ABB RAPID module: P6.mod

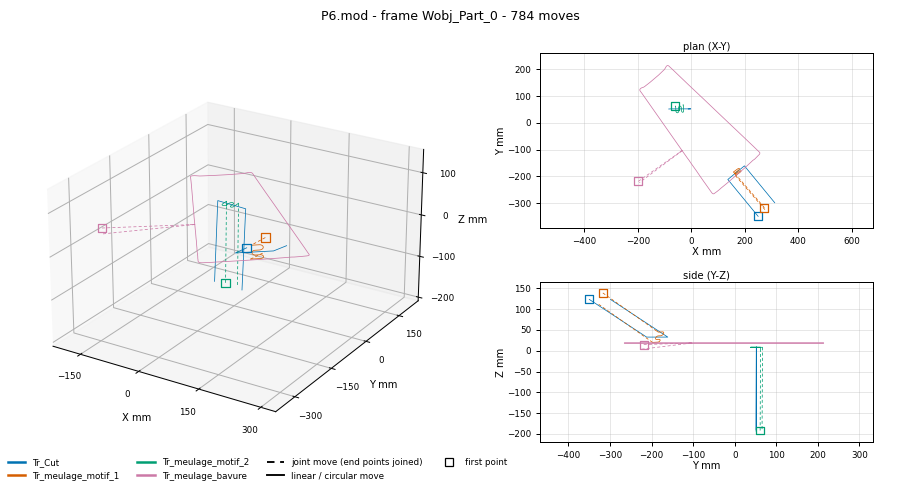
[picture p0: tool path of P6.mod in frame Wobj_Part_0, 784 of 794 moves have a stored position in this frame; points joined in program order, loops and branches not executed]
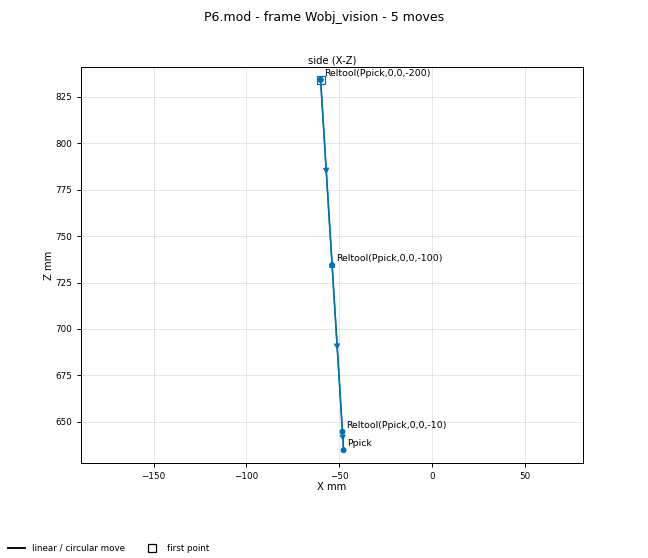
[picture p1: tool path of P6.mod in frame Wobj_vision, 5 of 794 moves have a stored position in this frame; points joined in program order, loops and branches not executed]
MODULE P6
	LOCAL CONST Speeddata vitesse_Tronconnage :=[10, 500, 0, 0];
	LOCAL CONST Robtarget Coupe_0 :=[[171.071296875,-183.16509375,32.79853125],[0.442625876519456,0.144946358690586,0.692091434062249,0.551436608718884],[0,0,0,0],[8.999999E+09,8.999999E+09,8.999999E+09,8.999999E+09,8.999999E+09,8.999999E+09]];
	LOCAL CONST Robtarget Coupe_1 :=[[-43.76221875,52.00546875,8.2563916015625],[0.723189251048334,-0.000890046614138083,-0.690648714177327,0.00093198196284652],[0,0,0,0],[8.999999E+09,8.999999E+09,8.999999E+09,8.999999E+09,8.999999E+09,8.999999E+09]];
	LOCAL CONST Robtarget Tr_meulage_motif_1_App1 :=[[272.919270252157,-317.055343641232,138.932114514029],[0.481869465480674,-0.803479210242735,-0.299818873825779,0.179809954793727],[0,0,0,0],[8.999999E+09,8.999999E+09,8.999999E+09,8.999999E+09,8.999999E+09,8.999999E+09]];
	LOCAL CONST Robtarget Tr_meulage_motif_1_App2 :=[[163.119364293858,-190.415905463312,49.4534391241389],[0.481869465480674,-0.803479210242735,-0.299818873825779,0.179809954793727],[0,0,0,0],[8.999999E+09,8.999999E+09,8.999999E+09,8.999999E+09,8.999999E+09,8.999999E+09]];
	LOCAL CONST Robtarget Tr_meulage_motif_1_P0 :=[[157.340421875,-183.750671875,44.74403515625],[0.481869465480674,-0.803479210242735,-0.299818873825779,0.179809954793727],[0,0,0,0],[8.999999E+09,8.999999E+09,8.999999E+09,8.999999E+09,8.999999E+09,8.999999E+09]];
	LOCAL CONST Robtarget Tr_meulage_motif_1_P1 :=[[158.144921875,-183.157578125,44.775765625],[0.481869465480674,-0.803479210242735,-0.299818873825779,0.179809954793727],[0,0,0,0],[8.999999E+09,8.999999E+09,8.999999E+09,8.999999E+09,8.999999E+09,8.999999E+09]];
	LOCAL CONST Robtarget Tr_meulage_motif_1_P2 :=[[158.949421875,-182.56446875,44.80749609375],[0.481869465480674,-0.803479210242735,-0.299818873825779,0.179809954793727],[0,0,0,0],[8.999999E+09,8.999999E+09,8.999999E+09,8.999999E+09,8.999999E+09,8.999999E+09]];
	LOCAL CONST Robtarget Tr_meulage_motif_1_P3 :=[[159.753921875,-181.971359375,44.8392265625],[0.481869465480674,-0.803479210242735,-0.299818873825779,0.179809954793727],[0,0,0,0],[8.999999E+09,8.999999E+09,8.999999E+09,8.999999E+09,8.999999E+09,8.999999E+09]];
	LOCAL CONST Robtarget Tr_meulage_motif_1_P4 :=[[160.558421875,-181.37825,44.87095703125],[0.481869465480674,-0.803479210242735,-0.299818873825779,0.179809954793727],[0,0,0,0],[8.999999E+09,8.999999E+09,8.999999E+09,8.999999E+09,8.999999E+09,8.999999E+09]];
	LOCAL CONST Robtarget Tr_meulage_motif_1_P5 :=[[161.362921875,-180.78515625,44.9026875],[0.481869465480674,-0.803479210242735,-0.299818873825779,0.179809954793727],[0,0,0,0],[8.999999E+09,8.999999E+09,8.999999E+09,8.999999E+09,8.999999E+09,8.999999E+09]];
	LOCAL CONST Robtarget Tr_meulage_motif_1_P6 :=[[162.167421875,-180.192046875,44.93441796875],[0.481869465480674,-0.803479210242735,-0.299818873825779,0.179809954793727],[0,0,0,0],[8.999999E+09,8.999999E+09,8.999999E+09,8.999999E+09,8.999999E+09,8.999999E+09]];
	LOCAL CONST Robtarget Tr_meulage_motif_1_P7 :=[[162.971921875,-179.5989375,44.9661484375],[0.481869465480674,-0.803479210242735,-0.299818873825779,0.179809954793727],[0,0,0,0],[8.999999E+09,8.999999E+09,8.999999E+09,8.999999E+09,8.999999E+09,8.999999E+09]];
	LOCAL CONST Robtarget Tr_meulage_motif_1_P8 :=[[163.776421875,-179.005828125,44.99787890625],[0.481869465480674,-0.803479210242735,-0.299818873825779,0.179809954793727],[0,0,0,0],[8.999999E+09,8.999999E+09,8.999999E+09,8.999999E+09,8.999999E+09,8.999999E+09]];
	LOCAL CONST Robtarget Tr_meulage_motif_1_P9 :=[[164.580921875,-178.412734375,45.029609375],[0.481869465480674,-0.803479210242735,-0.299818873825779,0.179809954793727],[0,0,0,0],[8.999999E+09,8.999999E+09,8.999999E+09,8.999999E+09,8.999999E+09,8.999999E+09]];
	LOCAL CONST Robtarget Tr_meulage_motif_1_P10 :=[[165.385421875,-177.819625,45.06133984375],[0.481869465480674,-0.803479210242735,-0.299818873825779,0.179809954793727],[0,0,0,0],[8.999999E+09,8.999999E+09,8.999999E+09,8.999999E+09,8.999999E+09,8.999999E+09]];
	LOCAL CONST Robtarget Tr_meulage_motif_1_P11 :=[[166.189921875,-177.226515625,45.0930703125],[0.481869465480674,-0.803479210242735,-0.299818873825779,0.179809954793727],[0,0,0,0],[8.999999E+09,8.999999E+09,8.999999E+09,8.999999E+09,8.999999E+09,8.999999E+09]];
	LOCAL CONST Robtarget Tr_meulage_motif_1_P12 :=[[166.994421875,-176.633421875,45.12480078125],[0.481869465480674,-0.803479210242735,-0.299818873825779,0.179809954793727],[0,0,0,0],[8.999999E+09,8.999999E+09,8.999999E+09,8.999999E+09,8.999999E+09,8.999999E+09]];
	LOCAL CONST Robtarget Tr_meulage_motif_1_P13 :=[[167.798921875,-176.0403125,45.15653125],[0.481869465480674,-0.803479210242735,-0.299818873825779,0.179809954793727],[0,0,0,0],[8.999999E+09,8.999999E+09,8.999999E+09,8.999999E+09,8.999999E+09,8.999999E+09]];
	LOCAL CONST Robtarget Tr_meulage_motif_1_P14 :=[[168.603421875,-175.447203125,45.18826171875],[0.481869465480674,-0.803479210242735,-0.299818873825779,0.179809954793727],[0,0,0,0],[8.999999E+09,8.999999E+09,8.999999E+09,8.999999E+09,8.999999E+09,8.999999E+09]];
	LOCAL CONST Robtarget Tr_meulage_motif_1_P15 :=[[169.407921875,-174.85409375,45.2199921875],[0.481869465480674,-0.803479210242735,-0.299818873825779,0.179809954793727],[0,0,0,0],[8.999999E+09,8.999999E+09,8.999999E+09,8.999999E+09,8.999999E+09,8.999999E+09]];
	LOCAL CONST Robtarget Tr_meulage_motif_1_P16 :=[[170.212421875,-174.261,45.25172265625],[0.481869465480674,-0.803479210242735,-0.299818873825779,0.179809954793727],[0,0,0,0],[8.999999E+09,8.999999E+09,8.999999E+09,8.999999E+09,8.999999E+09,8.999999E+09]];
	LOCAL CONST Robtarget Tr_meulage_motif_1_P17 :=[[171.016921875,-173.667890625,45.28345703125],[0.481869465480674,-0.803479210242735,-0.299818873825779,0.179809954793727],[0,0,0,0],[8.999999E+09,8.999999E+09,8.999999E+09,8.999999E+09,8.999999E+09,8.999999E+09]];
	LOCAL CONST Robtarget Tr_meulage_motif_1_P18 :=[[171.821421875,-173.07478125,45.3151875],[0.481869465480674,-0.803479210242735,-0.299818873825779,0.179809954793727],[0,0,0,0],[8.999999E+09,8.999999E+09,8.999999E+09,8.999999E+09,8.999999E+09,8.999999E+09]];
	LOCAL CONST Robtarget Tr_meulage_motif_1_P19 :=[[172.657078125,-172.531453125,45.25290625],[0.481869465480674,-0.803479210242735,-0.299818873825779,0.179809954793727],[0,0,0,0],[8.999999E+09,8.999999E+09,8.999999E+09,8.999999E+09,8.999999E+09,8.999999E+09]];
	LOCAL CONST Robtarget Tr_meulage_motif_1_P20 :=[[173.489453125,-172.0566875,45.1038671875],[0.481869465480674,-0.803479210242735,-0.299818873825779,0.179809954793727],[0,0,0,0],[8.999999E+09,8.999999E+09,8.999999E+09,8.999999E+09,8.999999E+09,8.999999E+09]];
	LOCAL CONST Robtarget Tr_meulage_motif_1_P21 :=[[174.26675,-171.6624375,44.90041796875],[0.481869465480674,-0.803479210242735,-0.299818873825779,0.179809954793727],[0,0,0,0],[8.999999E+09,8.999999E+09,8.999999E+09,8.999999E+09,8.999999E+09,8.999999E+09]];
	LOCAL CONST Robtarget Tr_meulage_motif_1_P22 :=[[174.96275,-171.330828125,44.69023828125],[0.481869465480674,-0.803479210242735,-0.299818873825779,0.179809954793727],[0,0,0,0],[8.999999E+09,8.999999E+09,8.999999E+09,8.999999E+09,8.999999E+09,8.999999E+09]];
	LOCAL CONST Robtarget Tr_meulage_motif_1_P23 :=[[176.05546875,-170.9305,44.2027421875],[0.481869465480674,-0.803479210242735,-0.299818873825779,0.179809954793727],[0,0,0,0],[8.999999E+09,8.999999E+09,8.999999E+09,8.999999E+09,8.999999E+09,8.999999E+09]];
	LOCAL CONST Robtarget Tr_meulage_motif_1_P24 :=[[177.16384375,-170.67090625,43.5164765625],[0.481869465480674,-0.803479210242735,-0.299818873825779,0.179809954793727],[0,0,0,0],[8.999999E+09,8.999999E+09,8.999999E+09,8.999999E+09,8.999999E+09,8.999999E+09]];
	LOCAL CONST Robtarget Tr_meulage_motif_1_P25 :=[[178.189625,-170.588109375,42.67519921875],[0.481869465480674,-0.803479210242735,-0.299818873825779,0.179809954793727],[0,0,0,0],[8.999999E+09,8.999999E+09,8.999999E+09,8.999999E+09,8.999999E+09,8.999999E+09]];
	LOCAL CONST Robtarget Tr_meulage_motif_1_P26 :=[[178.9571875,-170.756390625,41.74423828125],[0.481869465480674,-0.803479210242735,-0.299818873825779,0.179809954793727],[0,0,0,0],[8.999999E+09,8.999999E+09,8.999999E+09,8.999999E+09,8.999999E+09,8.999999E+09]];
	LOCAL CONST Robtarget Tr_meulage_motif_1_P27 :=[[179.2126875,-171.025796875,41.1549609375],[0.481869465480674,-0.803479210242735,-0.299818873825779,0.179809954793727],[0,0,0,0],[8.999999E+09,8.999999E+09,8.999999E+09,8.999999E+09,8.999999E+09,8.999999E+09]];
	LOCAL CONST Robtarget Tr_meulage_motif_1_P28 :=[[179.43475,-171.297015625,40.594265625],[0.481869465480674,-0.803479210242735,-0.299818873825779,0.179809954793727],[0,0,0,0],[8.999999E+09,8.999999E+09,8.999999E+09,8.999999E+09,8.999999E+09,8.999999E+09]];
	LOCAL CONST Robtarget Tr_meulage_motif_1_P29 :=[[179.612625,-171.60071875,40.03196484375],[0.481869465480674,-0.803479210242735,-0.299818873825779,0.179809954793727],[0,0,0,0],[8.999999E+09,8.999999E+09,8.999999E+09,8.999999E+09,8.999999E+09,8.999999E+09]];
	LOCAL CONST Robtarget Tr_meulage_motif_1_P30 :=[[179.5818125,-172.348109375,39.0819453125],[0.481869465480674,-0.803479210242735,-0.299818873825779,0.179809954793727],[0,0,0,0],[8.999999E+09,8.999999E+09,8.999999E+09,8.999999E+09,8.999999E+09,8.999999E+09]];
	LOCAL CONST Robtarget Tr_meulage_motif_1_P31 :=[[179.230703125,-173.2690625,38.20121484375],[0.481869465480674,-0.803479210242735,-0.299818873825779,0.179809954793727],[0,0,0,0],[8.999999E+09,8.999999E+09,8.999999E+09,8.999999E+09,8.999999E+09,8.999999E+09]];
	LOCAL CONST Robtarget Tr_meulage_motif_1_P32 :=[[178.685734375,-174.216015625,37.4659140625],[0.481869465480674,-0.803479210242735,-0.299818873825779,0.179809954793727],[0,0,0,0],[8.999999E+09,8.999999E+09,8.999999E+09,8.999999E+09,8.999999E+09,8.999999E+09]];
	LOCAL CONST Robtarget Tr_meulage_motif_1_P33 :=[[178.265875,-174.785859375,37.10854296875],[0.481869465480674,-0.803479210242735,-0.299818873825779,0.179809954793727],[0,0,0,0],[8.999999E+09,8.999999E+09,8.999999E+09,8.999999E+09,8.999999E+09,8.999999E+09]];
	LOCAL CONST Robtarget Tr_meulage_motif_1_P34 :=[[177.497859375,-175.672734375,36.6583984375],[0.481869465480674,-0.803479210242735,-0.299818873825779,0.179809954793727],[0,0,0,0],[8.999999E+09,8.999999E+09,8.999999E+09,8.999999E+09,8.999999E+09,8.999999E+09]];
	LOCAL CONST Robtarget Tr_meulage_motif_1_P35 :=[[176.906734375,-176.28225,36.40765234375],[0.481869465480674,-0.803479210242735,-0.299818873825779,0.179809954793727],[0,0,0,0],[8.999999E+09,8.999999E+09,8.999999E+09,8.999999E+09,8.999999E+09,8.999999E+09]];
	LOCAL CONST Robtarget Tr_meulage_motif_1_P36 :=[[176.22559375,-176.918890625,36.204703125],[0.481869465480674,-0.803479210242735,-0.299818873825779,0.179809954793727],[0,0,0,0],[8.999999E+09,8.999999E+09,8.999999E+09,8.999999E+09,8.999999E+09,8.999999E+09]];
	LOCAL CONST Robtarget Tr_meulage_motif_1_P37 :=[[175.47240625,-177.54559375,36.08148046875],[0.481869465480674,-0.803479210242735,-0.299818873825779,0.179809954793727],[0,0,0,0],[8.999999E+09,8.999999E+09,8.999999E+09,8.999999E+09,8.999999E+09,8.999999E+09]];
	LOCAL CONST Robtarget Tr_meulage_motif_1_P38 :=[[174.71103125,-178.17965625,35.95620703125],[0.481869465480674,-0.803479210242735,-0.299818873825779,0.179809954793727],[0,0,0,0],[8.999999E+09,8.999999E+09,8.999999E+09,8.999999E+09,8.999999E+09,8.999999E+09]];
	LOCAL CONST Robtarget Tr_meulage_motif_1_P39 :=[[173.90653125,-178.77275,35.9244765625],[0.481869465480674,-0.803479210242735,-0.299818873825779,0.179809954793727],[0,0,0,0],[8.999999E+09,8.999999E+09,8.999999E+09,8.999999E+09,8.999999E+09,8.999999E+09]];
	LOCAL CONST Robtarget Tr_meulage_motif_1_P40 :=[[173.10203125,-179.365859375,35.89274609375],[0.481869465480674,-0.803479210242735,-0.299818873825779,0.179809954793727],[0,0,0,0],[8.999999E+09,8.999999E+09,8.999999E+09,8.999999E+09,8.999999E+09,8.999999E+09]];
	LOCAL CONST Robtarget Tr_meulage_motif_1_P41 :=[[172.29753125,-179.95896875,35.861015625],[0.481869465480674,-0.803479210242735,-0.299818873825779,0.179809954793727],[0,0,0,0],[8.999999E+09,8.999999E+09,8.999999E+09,8.999999E+09,8.999999E+09,8.999999E+09]];
	LOCAL CONST Robtarget Tr_meulage_motif_1_P42 :=[[171.49303125,-180.552078125,35.82928515625],[0.481869465480674,-0.803479210242735,-0.299818873825779,0.179809954793727],[0,0,0,0],[8.999999E+09,8.999999E+09,8.999999E+09,8.999999E+09,8.999999E+09,8.999999E+09]];
	LOCAL CONST Robtarget Tr_meulage_motif_1_P43 :=[[170.68853125,-181.145171875,35.7975546875],[0.481869465480674,-0.803479210242735,-0.299818873825779,0.179809954793727],[0,0,0,0],[8.999999E+09,8.999999E+09,8.999999E+09,8.999999E+09,8.999999E+09,8.999999E+09]];
	LOCAL CONST Robtarget Tr_meulage_motif_1_P44 :=[[169.88403125,-181.73828125,35.76582421875],[0.481869465480674,-0.803479210242735,-0.299818873825779,0.179809954793727],[0,0,0,0],[8.999999E+09,8.999999E+09,8.999999E+09,8.999999E+09,8.999999E+09,8.999999E+09]];
	LOCAL CONST Robtarget Tr_meulage_motif_1_P45 :=[[169.07953125,-182.331390625,35.73409375],[0.481869465480674,-0.803479210242735,-0.299818873825779,0.179809954793727],[0,0,0,0],[8.999999E+09,8.999999E+09,8.999999E+09,8.999999E+09,8.999999E+09,8.999999E+09]];
	LOCAL CONST Robtarget Tr_meulage_motif_1_P46 :=[[168.27503125,-182.9245,35.70236328125],[0.481869465480674,-0.803479210242735,-0.299818873825779,0.179809954793727],[0,0,0,0],[8.999999E+09,8.999999E+09,8.999999E+09,8.999999E+09,8.999999E+09,8.999999E+09]];
	LOCAL CONST Robtarget Tr_meulage_motif_1_P47 :=[[167.47053125,-183.51759375,35.6706328125],[0.481869465480674,-0.803479210242735,-0.299818873825779,0.179809954793727],[0,0,0,0],[8.999999E+09,8.999999E+09,8.999999E+09,8.999999E+09,8.999999E+09,8.999999E+09]];
	LOCAL CONST Robtarget Tr_meulage_motif_1_P48 :=[[166.66603125,-184.110703125,35.63890234375],[0.481869465480674,-0.803479210242735,-0.299818873825779,0.179809954793727],[0,0,0,0],[8.999999E+09,8.999999E+09,8.999999E+09,8.999999E+09,8.999999E+09,8.999999E+09]];
	LOCAL CONST Robtarget Tr_meulage_motif_1_P49 :=[[165.90465625,-184.744765625,35.51362890625],[0.481869465480674,-0.803479210242735,-0.299818873825779,0.179809954793727],[0,0,0,0],[8.999999E+09,8.999999E+09,8.999999E+09,8.999999E+09,8.999999E+09,8.999999E+09]];
	LOCAL CONST Robtarget Tr_meulage_motif_1_P50 :=[[165.214125,-185.39275,35.3045234375],[0.481869465480674,-0.803479210242735,-0.299818873825779,0.179809954793727],[0,0,0,0],[8.999999E+09,8.999999E+09,8.999999E+09,8.999999E+09,8.999999E+09,8.999999E+09]];
	LOCAL CONST Robtarget Tr_meulage_motif_1_P51 :=[[164.61940625,-186.01,35.0469609375],[0.481869465480674,-0.803479210242735,-0.299818873825779,0.179809954793727],[0,0,0,0],[8.999999E+09,8.999999E+09,8.999999E+09,8.999999E+09,8.999999E+09,8.999999E+09]];
	LOCAL CONST Robtarget Tr_meulage_motif_1_P52 :=[[164.149140625,-186.55675,34.76648046875],[0.481869465480674,-0.803479210242735,-0.299818873825779,0.179809954793727],[0,0,0,0],[8.999999E+09,8.999999E+09,8.999999E+09,8.999999E+09,8.999999E+09,8.999999E+09]];
	LOCAL CONST Robtarget Tr_meulage_motif_1_P53 :=[[163.539421875,-187.442046875,34.171875],[0.481869465480674,-0.803479210242735,-0.299818873825779,0.179809954793727],[0,0,0,0],[8.999999E+09,8.999999E+09,8.999999E+09,8.999999E+09,8.999999E+09,8.999999E+09]];
	LOCAL CONST Robtarget Tr_meulage_motif_1_P54 :=[[163.116703125,-188.346921875,33.3784765625],[0.481869465480674,-0.803479210242735,-0.299818873825779,0.179809954793727],[0,0,0,0],[8.999999E+09,8.999999E+09,8.999999E+09,8.999999E+09,8.999999E+09,8.999999E+09]];
	LOCAL CONST Robtarget Tr_meulage_motif_1_P55 :=[[163.037609375,-189.093265625,32.4745390625],[0.481869465480674,-0.803479210242735,-0.299818873825779,0.179809954793727],[0,0,0,0],[8.999999E+09,8.999999E+09,8.999999E+09,8.999999E+09,8.999999E+09,8.999999E+09]];
	LOCAL CONST Robtarget Tr_meulage_motif_1_P56 :=[[163.12175,-189.4871875,31.880873046875],[0.481869465480674,-0.803479210242735,-0.299818873825779,0.179809954793727],[0,0,0,0],[8.999999E+09,8.999999E+09,8.999999E+09,8.999999E+09,8.999999E+09,8.999999E+09]];
	LOCAL CONST Robtarget Tr_meulage_motif_1_P57 :=[[163.328984375,-189.840875,31.225939453125],[0.481869465480674,-0.803479210242735,-0.299818873825779,0.179809954793727],[0,0,0,0],[8.999999E+09,8.999999E+09,8.999999E+09,8.999999E+09,8.999999E+09,8.999999E+09]];
	LOCAL CONST Robtarget Tr_meulage_motif_1_P58 :=[[163.641375,-190.116953125,30.57526171875],[0.481869465480674,-0.803479210242735,-0.299818873825779,0.179809954793727],[0,0,0,0],[8.999999E+09,8.999999E+09,8.999999E+09,8.999999E+09,8.999999E+09,8.999999E+09]];
	LOCAL CONST Robtarget Tr_meulage_motif_1_P59 :=[[164.351125,-190.322640625,29.648857421875],[0.481869465480674,-0.803479210242735,-0.299818873825779,0.179809954793727],[0,0,0,0],[8.999999E+09,8.999999E+09,8.999999E+09,8.999999E+09,8.999999E+09,8.999999E+09]];
	LOCAL CONST Robtarget Tr_meulage_motif_1_P60 :=[[164.881125,-190.317140625,29.165380859375],[0.481869465480674,-0.803479210242735,-0.299818873825779,0.179809954793727],[0,0,0,0],[8.999999E+09,8.999999E+09,8.999999E+09,8.999999E+09,8.999999E+09,8.999999E+09]];
	LOCAL CONST Robtarget Tr_meulage_motif_1_P61 :=[[165.892734375,-190.15484375,28.44130859375],[0.481869465480674,-0.803479210242735,-0.299818873825779,0.179809954793727],[0,0,0,0],[8.999999E+09,8.999999E+09,8.999999E+09,8.999999E+09,8.999999E+09,8.999999E+09]];
	LOCAL CONST Robtarget Tr_meulage_motif_1_P62 :=[[166.5030625,-189.97740625,28.108583984375],[0.481869465480674,-0.803479210242735,-0.299818873825779,0.179809954793727],[0,0,0,0],[8.999999E+09,8.999999E+09,8.999999E+09,8.999999E+09,8.999999E+09,8.999999E+09]];
	LOCAL CONST Robtarget Tr_meulage_motif_1_P63 :=[[167.585140625,-189.53753125,27.682701171875],[0.481869465480674,-0.803479210242735,-0.299818873825779,0.179809954793727],[0,0,0,0],[8.999999E+09,8.999999E+09,8.999999E+09,8.999999E+09,8.999999E+09,8.999999E+09]];
	LOCAL CONST Robtarget Tr_meulage_motif_1_P64 :=[[168.3485625,-189.169078125,27.458333984375],[0.481869465480674,-0.803479210242735,-0.299818873825779,0.179809954793727],[0,0,0,0],[8.999999E+09,8.999999E+09,8.999999E+09,8.999999E+09,8.999999E+09,8.999999E+09]];
	LOCAL CONST Robtarget Tr_meulage_motif_1_P65 :=[[169.16703125,-188.70015625,27.31453125],[0.481869465480674,-0.803479210242735,-0.299818873825779,0.179809954793727],[0,0,0,0],[8.999999E+09,8.999999E+09,8.999999E+09,8.999999E+09,8.999999E+09,8.999999E+09]];
	LOCAL CONST Robtarget Tr_meulage_motif_1_P66 :=[[169.99315625,-188.16253125,27.25359765625],[0.481869465480674,-0.803479210242735,-0.299818873825779,0.179809954793727],[0,0,0,0],[8.999999E+09,8.999999E+09,8.999999E+09,8.999999E+09,8.999999E+09,8.999999E+09]];
	LOCAL CONST Robtarget Tr_meulage_motif_1_P67 :=[[170.8288125,-187.619203125,27.19131640625],[0.481869465480674,-0.803479210242735,-0.299818873825779,0.179809954793727],[0,0,0,0],[8.999999E+09,8.999999E+09,8.999999E+09,8.999999E+09,8.999999E+09,8.999999E+09]];
	LOCAL CONST Robtarget Tr_meulage_motif_1_P68 :=[[171.6333125,-187.02609375,27.223046875],[0.481869465480674,-0.803479210242735,-0.299818873825779,0.179809954793727],[0,0,0,0],[8.999999E+09,8.999999E+09,8.999999E+09,8.999999E+09,8.999999E+09,8.999999E+09]];
	LOCAL CONST Robtarget Tr_meulage_motif_1_P69 :=[[172.4378125,-186.432984375,27.25477734375],[0.481869465480674,-0.803479210242735,-0.299818873825779,0.179809954793727],[0,0,0,0],[8.999999E+09,8.999999E+09,8.999999E+09,8.999999E+09,8.999999E+09,8.999999E+09]];
	LOCAL CONST Robtarget Tr_meulage_motif_1_P70 :=[[173.2423125,-185.839890625,27.2865078125],[0.481869465480674,-0.803479210242735,-0.299818873825779,0.179809954793727],[0,0,0,0],[8.999999E+09,8.999999E+09,8.999999E+09,8.999999E+09,8.999999E+09,8.999999E+09]];
	LOCAL CONST Robtarget Tr_meulage_motif_1_P71 :=[[174.0468125,-185.24678125,27.31823828125],[0.481869465480674,-0.803479210242735,-0.299818873825779,0.179809954793727],[0,0,0,0],[8.999999E+09,8.999999E+09,8.999999E+09,8.999999E+09,8.999999E+09,8.999999E+09]];
	LOCAL CONST Robtarget Tr_meulage_motif_1_P72 :=[[174.8513125,-184.653671875,27.34996875],[0.481869465480674,-0.803479210242735,-0.299818873825779,0.179809954793727],[0,0,0,0],[8.999999E+09,8.999999E+09,8.999999E+09,8.999999E+09,8.999999E+09,8.999999E+09]];
	LOCAL CONST Robtarget Tr_meulage_motif_1_P73 :=[[175.6558125,-184.0605625,27.38169921875],[0.481869465480674,-0.803479210242735,-0.299818873825779,0.179809954793727],[0,0,0,0],[8.999999E+09,8.999999E+09,8.999999E+09,8.999999E+09,8.999999E+09,8.999999E+09]];
	LOCAL CONST Robtarget Tr_meulage_motif_1_P74 :=[[176.4603125,-183.46746875,27.413431640625],[0.481869465480674,-0.803479210242735,-0.299818873825779,0.179809954793727],[0,0,0,0],[8.999999E+09,8.999999E+09,8.999999E+09,8.999999E+09,8.999999E+09,8.999999E+09]];
	LOCAL CONST Robtarget Tr_meulage_motif_1_P75 :=[[177.2648125,-182.874359375,27.445162109375],[0.481869465480674,-0.803479210242735,-0.299818873825779,0.179809954793727],[0,0,0,0],[8.999999E+09,8.999999E+09,8.999999E+09,8.999999E+09,8.999999E+09,8.999999E+09]];
	LOCAL CONST Robtarget Tr_meulage_motif_1_P76 :=[[178.0693125,-182.28125,27.476892578125],[0.481869465480674,-0.803479210242735,-0.299818873825779,0.179809954793727],[0,0,0,0],[8.999999E+09,8.999999E+09,8.999999E+09,8.999999E+09,8.999999E+09,8.999999E+09]];
	LOCAL CONST Robtarget Tr_meulage_motif_1_P77 :=[[178.8738125,-181.688140625,27.508623046875],[0.481869465480674,-0.803479210242735,-0.299818873825779,0.179809954793727],[0,0,0,0],[8.999999E+09,8.999999E+09,8.999999E+09,8.999999E+09,8.999999E+09,8.999999E+09]];
	LOCAL CONST Robtarget Tr_meulage_motif_1_P78 :=[[179.70946875,-181.1448125,27.446341796875],[0.481869465480674,-0.803479210242735,-0.299818873825779,0.179809954793727],[0,0,0,0],[8.999999E+09,8.999999E+09,8.999999E+09,8.999999E+09,8.999999E+09,8.999999E+09]];
	LOCAL CONST Robtarget Tr_meulage_motif_1_P79 :=[[180.54184375,-180.6700625,27.297302734375],[0.481869465480674,-0.803479210242735,-0.299818873825779,0.179809954793727],[0,0,0,0],[8.999999E+09,8.999999E+09,8.999999E+09,8.999999E+09,8.999999E+09,8.999999E+09]];
	LOCAL CONST Robtarget Tr_meulage_motif_1_P80 :=[[181.31915625,-180.2758125,27.09385546875],[0.481869465480674,-0.803479210242735,-0.299818873825779,0.179809954793727],[0,0,0,0],[8.999999E+09,8.999999E+09,8.999999E+09,8.999999E+09,8.999999E+09,8.999999E+09]];
	LOCAL CONST Robtarget Tr_meulage_motif_1_P81 :=[[182.015140625,-179.9441875,26.883673828125],[0.481869465480674,-0.803479210242735,-0.299818873825779,0.179809954793727],[0,0,0,0],[8.999999E+09,8.999999E+09,8.999999E+09,8.999999E+09,8.999999E+09,8.999999E+09]];
	LOCAL CONST Robtarget Tr_meulage_motif_1_P82 :=[[183.107859375,-179.543859375,26.3961796875],[0.481869465480674,-0.803479210242735,-0.299818873825779,0.179809954793727],[0,0,0,0],[8.999999E+09,8.999999E+09,8.999999E+09,8.999999E+09,8.999999E+09,8.999999E+09]];
	LOCAL CONST Robtarget Tr_meulage_motif_1_P83 :=[[184.177765625,-179.34309375,25.668513671875],[0.481869465480674,-0.803479210242735,-0.299818873825779,0.179809954793727],[0,0,0,0],[8.999999E+09,8.999999E+09,8.999999E+09,8.999999E+09,8.999999E+09,8.999999E+09]];
	LOCAL CONST Robtarget Tr_meulage_motif_1_P84 :=[[185.032515625,-179.42725,24.76698828125],[0.481869465480674,-0.803479210242735,-0.299818873825779,0.179809954793727],[0,0,0,0],[8.999999E+09,8.999999E+09,8.999999E+09,8.999999E+09,8.999999E+09,8.999999E+09]];
	LOCAL CONST Robtarget Tr_meulage_motif_1_P85 :=[[185.499296875,-179.730578125,23.937677734375],[0.481869465480674,-0.803479210242735,-0.299818873825779,0.179809954793727],[0,0,0,0],[8.999999E+09,8.999999E+09,8.999999E+09,8.999999E+09,8.999999E+09,8.999999E+09]];
	LOCAL CONST Robtarget Tr_meulage_motif_1_P86 :=[[185.462265625,-179.8925,23.759970703125],[0.481869465480674,-0.803479210242735,-0.299818873825779,0.179809954793727],[0,0,0,0],[8.999999E+09,8.999999E+09,8.999999E+09,8.999999E+09,8.999999E+09,8.999999E+09]];
	LOCAL CONST Robtarget Tr_meulage_motif_1_P87 :=[[185.606953125,-180.263609375,23.14011328125],[0.481869465480674,-0.803479210242735,-0.299818873825779,0.179809954793727],[0,0,0,0],[8.999999E+09,8.999999E+09,8.999999E+09,8.999999E+09,8.999999E+09,8.999999E+09]];
	LOCAL CONST Robtarget Tr_meulage_motif_1_P88 :=[[185.371328125,-181.053578125,22.3239765625],[0.481869465480674,-0.803479210242735,-0.299818873825779,0.179809954793727],[0,0,0,0],[8.999999E+09,8.999999E+09,8.999999E+09,8.999999E+09,8.999999E+09,8.999999E+09]];
	LOCAL CONST Robtarget Tr_meulage_motif_1_P89 :=[[185.07846875,-181.574546875,21.913001953125],[0.481869465480674,-0.803479210242735,-0.299818873825779,0.179809954793727],[0,0,0,0],[8.999999E+09,8.999999E+09,8.999999E+09,8.999999E+09,8.999999E+09,8.999999E+09]];
	LOCAL CONST Robtarget Tr_meulage_motif_1_P90 :=[[184.34728125,-182.462515625,21.427361328125],[0.481869465480674,-0.803479210242735,-0.299818873825779,0.179809954793727],[0,0,0,0],[8.999999E+09,8.999999E+09,8.999999E+09,8.999999E+09,8.999999E+09,8.999999E+09]];
	LOCAL CONST Robtarget Tr_meulage_motif_1_P91 :=[[183.756140625,-183.072015625,21.176615234375],[0.481869465480674,-0.803479210242735,-0.299818873825779,0.179809954793727],[0,0,0,0],[8.999999E+09,8.999999E+09,8.999999E+09,8.999999E+09,8.999999E+09,8.999999E+09]];
	LOCAL CONST Robtarget Tr_meulage_motif_1_P92 :=[[183.075015625,-183.70865625,20.973666015625],[0.481869465480674,-0.803479210242735,-0.299818873825779,0.179809954793727],[0,0,0,0],[8.999999E+09,8.999999E+09,8.999999E+09,8.999999E+09,8.999999E+09,8.999999E+09]];
	LOCAL CONST Robtarget Tr_meulage_motif_1_P93 :=[[182.3218125,-184.335375,20.85044140625],[0.481869465480674,-0.803479210242735,-0.299818873825779,0.179809954793727],[0,0,0,0],[8.999999E+09,8.999999E+09,8.999999E+09,8.999999E+09,8.999999E+09,8.999999E+09]];
	LOCAL CONST Robtarget Tr_meulage_motif_1_P94 :=[[181.5604375,-184.969421875,20.725169921875],[0.481869465480674,-0.803479210242735,-0.299818873825779,0.179809954793727],[0,0,0,0],[8.999999E+09,8.999999E+09,8.999999E+09,8.999999E+09,8.999999E+09,8.999999E+09]];
	LOCAL CONST Robtarget Tr_meulage_motif_1_P95 :=[[180.7559375,-185.56253125,20.693439453125],[0.481869465480674,-0.803479210242735,-0.299818873825779,0.179809954793727],[0,0,0,0],[8.999999E+09,8.999999E+09,8.999999E+09,8.999999E+09,8.999999E+09,8.999999E+09]];
	LOCAL CONST Robtarget Tr_meulage_motif_1_P96 :=[[179.9514375,-186.155640625,20.661708984375],[0.481869465480674,-0.803479210242735,-0.299818873825779,0.179809954793727],[0,0,0,0],[8.999999E+09,8.999999E+09,8.999999E+09,8.999999E+09,8.999999E+09,8.999999E+09]];
	LOCAL CONST Robtarget Tr_meulage_motif_1_P97 :=[[179.1469375,-186.74875,20.629978515625],[0.481869465480674,-0.803479210242735,-0.299818873825779,0.179809954793727],[0,0,0,0],[8.999999E+09,8.999999E+09,8.999999E+09,8.999999E+09,8.999999E+09,8.999999E+09]];
	LOCAL CONST Robtarget Tr_meulage_motif_1_P98 :=[[178.3424375,-187.34184375,20.598248046875],[0.481869465480674,-0.803479210242735,-0.299818873825779,0.179809954793727],[0,0,0,0],[8.999999E+09,8.999999E+09,8.999999E+09,8.999999E+09,8.999999E+09,8.999999E+09]];
	LOCAL CONST Robtarget Tr_meulage_motif_1_P99 :=[[177.5379375,-187.934953125,20.566517578125],[0.481869465480674,-0.803479210242735,-0.299818873825779,0.179809954793727],[0,0,0,0],[8.999999E+09,8.999999E+09,8.999999E+09,8.999999E+09,8.999999E+09,8.999999E+09]];
	LOCAL CONST Robtarget Tr_meulage_motif_1_P100 :=[[176.7334375,-188.5280625,20.534787109375],[0.481869465480674,-0.803479210242735,-0.299818873825779,0.179809954793727],[0,0,0,0],[8.999999E+09,8.999999E+09,8.999999E+09,8.999999E+09,8.999999E+09,8.999999E+09]];
	LOCAL CONST Robtarget Tr_meulage_motif_1_P101 :=[[175.9289375,-189.121171875,20.5030546875],[0.481869465480674,-0.803479210242735,-0.299818873825779,0.179809954793727],[0,0,0,0],[8.999999E+09,8.999999E+09,8.999999E+09,8.999999E+09,8.999999E+09,8.999999E+09]];
	LOCAL CONST Robtarget Tr_meulage_motif_1_P102 :=[[175.1244375,-189.714265625,20.47132421875],[0.481869465480674,-0.803479210242735,-0.299818873825779,0.179809954793727],[0,0,0,0],[8.999999E+09,8.999999E+09,8.999999E+09,8.999999E+09,8.999999E+09,8.999999E+09]];
	LOCAL CONST Robtarget Tr_meulage_motif_1_P103 :=[[174.3199375,-190.307375,20.43959375],[0.481869465480674,-0.803479210242735,-0.299818873825779,0.179809954793727],[0,0,0,0],[8.999999E+09,8.999999E+09,8.999999E+09,8.999999E+09,8.999999E+09,8.999999E+09]];
	LOCAL CONST Robtarget Tr_meulage_motif_1_P104 :=[[173.5154375,-190.900484375,20.40786328125],[0.481869465480674,-0.803479210242735,-0.299818873825779,0.179809954793727],[0,0,0,0],[8.999999E+09,8.999999E+09,8.999999E+09,8.999999E+09,8.999999E+09,8.999999E+09]];
	LOCAL CONST Robtarget Tr_meulage_motif_1_P105 :=[[172.7109375,-191.49359375,20.3761328125],[0.481869465480674,-0.803479210242735,-0.299818873825779,0.179809954793727],[0,0,0,0],[8.999999E+09,8.999999E+09,8.999999E+09,8.999999E+09,8.999999E+09,8.999999E+09]];
	LOCAL CONST Robtarget Tr_meulage_motif_1_P106 :=[[171.9064375,-192.0866875,20.34440234375],[0.481869465480674,-0.803479210242735,-0.299818873825779,0.179809954793727],[0,0,0,0],[8.999999E+09,8.999999E+09,8.999999E+09,8.999999E+09,8.999999E+09,8.999999E+09]];
	LOCAL CONST Robtarget Tr_meulage_motif_1_P107 :=[[171.101953125,-192.679796875,20.312671875],[0.481869465480674,-0.803479210242735,-0.299818873825779,0.179809954793727],[0,0,0,0],[8.999999E+09,8.999999E+09,8.999999E+09,8.999999E+09,8.999999E+09,8.999999E+09]];
	LOCAL CONST Robtarget Tr_meulage_motif_1_P108 :=[[170.297453125,-193.27290625,20.28094140625],[0.481869465480674,-0.803479210242735,-0.299818873825779,0.179809954793727],[0,0,0,0],[8.999999E+09,8.999999E+09,8.999999E+09,8.999999E+09,8.999999E+09,8.999999E+09]];
	LOCAL CONST Robtarget Tr_meulage_motif_1_P109 :=[[169.492953125,-193.866,20.249208984375],[0.481869465480674,-0.803479210242735,-0.299818873825779,0.179809954793727],[0,0,0,0],[8.999999E+09,8.999999E+09,8.999999E+09,8.999999E+09,8.999999E+09,8.999999E+09]];
	LOCAL CONST Robtarget Tr_meulage_motif_1_P110 :=[[168.688453125,-194.459109375,20.217478515625],[0.481869465480674,-0.803479210242735,-0.299818873825779,0.179809954793727],[0,0,0,0],[8.999999E+09,8.999999E+09,8.999999E+09,8.999999E+09,8.999999E+09,8.999999E+09]];
	LOCAL CONST Robtarget Tr_meulage_motif_1_P111 :=[[167.883953125,-195.05221875,20.185748046875],[0.481869465480674,-0.803479210242735,-0.299818873825779,0.179809954793727],[0,0,0,0],[8.999999E+09,8.999999E+09,8.999999E+09,8.999999E+09,8.999999E+09,8.999999E+09]];
	LOCAL CONST Robtarget Tr_meulage_motif_1_P112 :=[[167.079453125,-195.645328125,20.154017578125],[0.481869465480674,-0.803479210242735,-0.299818873825779,0.179809954793727],[0,0,0,0],[8.999999E+09,8.999999E+09,8.999999E+09,8.999999E+09,8.999999E+09,8.999999E+09]];
	LOCAL CONST Robtarget Tr_meulage_motif_1_P113 :=[[166.274953125,-196.238421875,20.122287109375],[0.481869465480674,-0.803479210242735,-0.299818873825779,0.179809954793727],[0,0,0,0],[8.999999E+09,8.999999E+09,8.999999E+09,8.999999E+09,8.999999E+09,8.999999E+09]];
	LOCAL CONST Robtarget Tr_meulage_motif_1_P114 :=[[165.470453125,-196.83153125,20.090556640625],[0.481869465480674,-0.803479210242735,-0.299818873825779,0.179809954793727],[0,0,0,0],[8.999999E+09,8.999999E+09,8.999999E+09,8.999999E+09,8.999999E+09,8.999999E+09]];
	LOCAL CONST Robtarget Tr_meulage_motif_1_P115 :=[[164.665953125,-197.424640625,20.058826171875],[0.481869465480674,-0.803479210242735,-0.299818873825779,0.179809954793727],[0,0,0,0],[8.999999E+09,8.999999E+09,8.999999E+09,8.999999E+09,8.999999E+09,8.999999E+09]];
	LOCAL CONST Robtarget Tr_meulage_motif_1_degg1 :=[[170.444895543858,-204.089874213312,24.7682301397639],[0.481869465480674,-0.803479210242735,-0.299818873825779,0.179809954793727],[0,0,0,0],[8.999999E+09,8.999999E+09,8.999999E+09,8.999999E+09,8.999999E+09,8.999999E+09]];
	LOCAL CONST Robtarget Tr_meulage_motif_1_degg2 :=[[280.244801502157,-330.729312391232,114.246905529654],[0.481869465480674,-0.803479210242735,-0.299818873825779,0.179809954793727],[0,0,0,0],[8.999999E+09,8.999999E+09,8.999999E+09,8.999999E+09,8.999999E+09,8.999999E+09]];
	LOCAL CONST Robtarget Tr_meulage_motif_2_App1 :=[[-61.2100200325105,61.1357100750485,-191.721200011354],[-1.55313807294348E-05,0.00588516465292523,0.0026390183776894,0.99997919987257],[0,0,0,0],[8.999999E+09,8.999999E+09,8.999999E+09,8.999999E+09,8.999999E+09,8.999999E+09]];
	LOCAL CONST Robtarget Tr_meulage_motif_2_App2 :=[[-58.973719556313,62.1385509334399,-1.7370078521302],[-1.55313807294348E-05,0.00588516465292523,0.0026390183776894,0.99997919987257],[0,0,0,0],[8.999999E+09,8.999999E+09,8.999999E+09,8.999999E+09,8.999999E+09,8.999999E+09]];
	LOCAL CONST Robtarget Tr_meulage_motif_2_P0 :=[[-58.85601953125,62.19133203125,8.26216015625],[-1.55313807294348E-05,0.00588516465292523,0.0026390183776894,0.99997919987257],[0,0,0,0],[8.999999E+09,8.999999E+09,8.999999E+09,8.999999E+09,8.999999E+09,8.999999E+09]];
	LOCAL CONST Robtarget Tr_meulage_motif_2_P1 :=[[-58.80004296875,61.19290234375,8.2646171875],[-1.55313807294348E-05,0.00588516465292523,0.0026390183776894,0.99997919987257],[0,0,0,0],[8.999999E+09,8.999999E+09,8.999999E+09,8.999999E+09,8.999999E+09,8.999999E+09]];
	LOCAL CONST Robtarget Tr_meulage_motif_2_P2 :=[[-58.74406640625,60.19447265625,8.2670732421875],[-1.55313807294348E-05,0.00588516465292523,0.0026390183776894,0.99997919987257],[0,0,0,0],[8.999999E+09,8.999999E+09,8.999999E+09,8.999999E+09,8.999999E+09,8.999999E+09]];
	LOCAL CONST Robtarget Tr_meulage_motif_2_P3 :=[[-58.68808984375,59.19604296875,8.2695302734375],[-1.55313807294348E-05,0.00588516465292523,0.0026390183776894,0.99997919987257],[0,0,0,0],[8.999999E+09,8.999999E+09,8.999999E+09,8.999999E+09,8.999999E+09,8.999999E+09]];
	LOCAL CONST Robtarget Tr_meulage_motif_2_P4 :=[[-58.63211328125,58.1976171875,8.271986328125],[-1.55313807294348E-05,0.00588516465292523,0.0026390183776894,0.99997919987257],[0,0,0,0],[8.999999E+09,8.999999E+09,8.999999E+09,8.999999E+09,8.999999E+09,8.999999E+09]];
	LOCAL CONST Robtarget Tr_meulage_motif_2_P5 :=[[-58.57613671875,57.1991875,8.274443359375],[-1.55313807294348E-05,0.00588516465292523,0.0026390183776894,0.99997919987257],[0,0,0,0],[8.999999E+09,8.999999E+09,8.999999E+09,8.999999E+09,8.999999E+09,8.999999E+09]];
	LOCAL CONST Robtarget Tr_meulage_motif_2_P6 :=[[-58.52016015625,56.2007578125,8.2768994140625],[-1.55313807294348E-05,0.00588516465292523,0.0026390183776894,0.99997919987257],[0,0,0,0],[8.999999E+09,8.999999E+09,8.999999E+09,8.999999E+09,8.999999E+09,8.999999E+09]];
	LOCAL CONST Robtarget Tr_meulage_motif_2_P7 :=[[-58.46418359375,55.202328125,8.27935546875],[-1.55313807294348E-05,0.00588516465292523,0.0026390183776894,0.99997919987257],[0,0,0,0],[8.999999E+09,8.999999E+09,8.999999E+09,8.999999E+09,8.999999E+09,8.999999E+09]];
	LOCAL CONST Robtarget Tr_meulage_motif_2_P8 :=[[-58.40820703125,54.2038984375,8.2818125],[-1.55313807294348E-05,0.00588516465292523,0.0026390183776894,0.99997919987257],[0,0,0,0],[8.999999E+09,8.999999E+09,8.999999E+09,8.999999E+09,8.999999E+09,8.999999E+09]];
	LOCAL CONST Robtarget Tr_meulage_motif_2_P9 :=[[-58.35223046875,53.20546875,8.2842685546875],[-1.55313807294348E-05,0.00588516465292523,0.0026390183776894,0.99997919987257],[0,0,0,0],[8.999999E+09,8.999999E+09,8.999999E+09,8.999999E+09,8.999999E+09,8.999999E+09]];
	LOCAL CONST Robtarget Tr_meulage_motif_2_P10 :=[[-58.29625390625,52.20704296875,8.2867255859375],[-1.55313807294348E-05,0.00588516465292523,0.0026390183776894,0.99997919987257],[0,0,0,0],[8.999999E+09,8.999999E+09,8.999999E+09,8.999999E+09,8.999999E+09,8.999999E+09]];
	LOCAL CONST Robtarget Tr_meulage_motif_2_P11 :=[[-58.24027734375,51.20861328125,8.289181640625],[-1.55313807294348E-05,0.00588516465292523,0.0026390183776894,0.99997919987257],[0,0,0,0],[8.999999E+09,8.999999E+09,8.999999E+09,8.999999E+09,8.999999E+09,8.999999E+09]];
	LOCAL CONST Robtarget Tr_meulage_motif_2_P12 :=[[-58.18430078125,50.21018359375,8.291638671875],[-1.55313807294348E-05,0.00588516465292523,0.0026390183776894,0.99997919987257],[0,0,0,0],[8.999999E+09,8.999999E+09,8.999999E+09,8.999999E+09,8.999999E+09,8.999999E+09]];
	LOCAL CONST Robtarget Tr_meulage_motif_2_P13 :=[[-58.12832421875,49.21175390625,8.2940947265625],[-1.55313807294348E-05,0.00588516465292523,0.0026390183776894,0.99997919987257],[0,0,0,0],[8.999999E+09,8.999999E+09,8.999999E+09,8.999999E+09,8.999999E+09,8.999999E+09]];
	LOCAL CONST Robtarget Tr_meulage_motif_2_P14 :=[[-58.07234765625,48.21332421875,8.2965517578125],[-1.55313807294348E-05,0.00588516465292523,0.0026390183776894,0.99997919987257],[0,0,0,0],[8.999999E+09,8.999999E+09,8.999999E+09,8.999999E+09,8.999999E+09,8.999999E+09]];
	LOCAL CONST Robtarget Tr_meulage_motif_2_P15 :=[[-58.01637109375,47.21489453125,8.2990078125],[-1.55313807294348E-05,0.00588516465292523,0.0026390183776894,0.99997919987257],[0,0,0,0],[8.999999E+09,8.999999E+09,8.999999E+09,8.999999E+09,8.999999E+09,8.999999E+09]];
	LOCAL CONST Robtarget Tr_meulage_motif_2_P16 :=[[-57.96039453125,46.21646875,8.3014638671875],[-1.55313807294348E-05,0.00588516465292523,0.0026390183776894,0.99997919987257],[0,0,0,0],[8.999999E+09,8.999999E+09,8.999999E+09,8.999999E+09,8.999999E+09,8.999999E+09]];
	LOCAL CONST Robtarget Tr_meulage_motif_2_P17 :=[[-57.90441796875,45.2180390625,8.3039208984375],[-1.55313807294348E-05,0.00588516465292523,0.0026390183776894,0.99997919987257],[0,0,0,0],[8.999999E+09,8.999999E+09,8.999999E+09,8.999999E+09,8.999999E+09,8.999999E+09]];
	LOCAL CONST Robtarget Tr_meulage_motif_2_P18 :=[[-57.8484375,44.219609375,8.306376953125],[-1.55313807294348E-05,0.00588516465292523,0.0026390183776894,0.99997919987257],[0,0,0,0],[8.999999E+09,8.999999E+09,8.999999E+09,8.999999E+09,8.999999E+09,8.999999E+09]];
	LOCAL CONST Robtarget Tr_meulage_motif_2_P19 :=[[-57.68245703125,43.234796875,8.3085654296875],[-1.55313807294348E-05,0.00588516465292523,0.0026390183776894,0.99997919987257],[0,0,0,0],[8.999999E+09,8.999999E+09,8.999999E+09,8.999999E+09,8.999999E+09,8.999999E+09]];
	LOCAL CONST Robtarget Tr_meulage_motif_2_P20 :=[[-57.41862109375,42.3016015625,8.310412109375],[-1.55313807294348E-05,0.00588516465292523,0.0026390183776894,0.99997919987257],[0,0,0,0],[8.999999E+09,8.999999E+09,8.999999E+09,8.999999E+09,8.999999E+09,8.999999E+09]];
	LOCAL CONST Robtarget Tr_meulage_motif_2_P21 :=[[-57.09947265625,41.46544140625,8.3118916015625],[-1.55313807294348E-05,0.00588516465292523,0.0026390183776894,0.99997919987257],[0,0,0,0],[8.999999E+09,8.999999E+09,8.999999E+09,8.999999E+09,8.999999E+09,8.999999E+09]];
	LOCAL CONST Robtarget Tr_meulage_motif_2_P22 :=[[-56.78198828125,40.732125,8.313109375],[-1.55313807294348E-05,0.00588516465292523,0.0026390183776894,0.99997919987257],[0,0,0,0],[8.999999E+09,8.999999E+09,8.999999E+09,8.999999E+09,8.999999E+09,8.999999E+09]];
	LOCAL CONST Robtarget Tr_meulage_motif_2_P23 :=[[-56.1051953125,39.66727734375,8.3144189453125],[-1.55313807294348E-05,0.00588516465292523,0.0026390183776894,0.99997919987257],[0,0,0,0],[8.999999E+09,8.999999E+09,8.999999E+09,8.999999E+09,8.999999E+09,8.999999E+09]];
	LOCAL CONST Robtarget Tr_meulage_motif_2_P24 :=[[-55.20155859375,38.69245703125,8.3150146484375],[-1.55313807294348E-05,0.00588516465292523,0.0026390183776894,0.99997919987257],[0,0,0,0],[8.999999E+09,8.999999E+09,8.999999E+09,8.999999E+09,8.999999E+09,8.999999E+09]];
	LOCAL CONST Robtarget Tr_meulage_motif_2_P25 :=[[-54.13183984375,37.9034375,8.314779296875],[-1.55313807294348E-05,0.00588516465292523,0.0026390183776894,0.99997919987257],[0,0,0,0],[8.999999E+09,8.999999E+09,8.999999E+09,8.999999E+09,8.999999E+09,8.999999E+09]];
	LOCAL CONST Robtarget Tr_meulage_motif_2_P26 :=[[-52.99008203125,37.4785234375,8.313451171875],[-1.55313807294348E-05,0.00588516465292523,0.0026390183776894,0.99997919987257],[0,0,0,0],[8.999999E+09,8.999999E+09,8.999999E+09,8.999999E+09,8.999999E+09,8.999999E+09]];
	LOCAL CONST Robtarget Tr_meulage_motif_2_P27 :=[[-52.29369140625,37.49045703125,8.3119423828125],[-1.55313807294348E-05,0.00588516465292523,0.0026390183776894,0.99997919987257],[0,0,0,0],[8.999999E+09,8.999999E+09,8.999999E+09,8.999999E+09,8.999999E+09,8.999999E+09]];
	LOCAL CONST Robtarget Tr_meulage_motif_2_P28 :=[[-51.63348046875,37.52746875,8.3104453125],[-1.55313807294348E-05,0.00588516465292523,0.0026390183776894,0.99997919987257],[0,0,0,0],[8.999999E+09,8.999999E+09,8.999999E+09,8.999999E+09,8.999999E+09,8.999999E+09]];
	LOCAL CONST Robtarget Tr_meulage_motif_2_P29 :=[[-50.97649609375,37.6192578125,8.308814453125],[-1.55313807294348E-05,0.00588516465292523,0.0026390183776894,0.99997919987257],[0,0,0,0],[8.999999E+09,8.999999E+09,8.999999E+09,8.999999E+09,8.999999E+09,8.999999E+09]];
	LOCAL CONST Robtarget Tr_meulage_motif_2_P30 :=[[-49.90436328125,38.17836328125,8.305095703125],[-1.55313807294348E-05,0.00588516465292523,0.0026390183776894,0.99997919987257],[0,0,0,0],[8.999999E+09,8.999999E+09,8.999999E+09,8.999999E+09,8.999999E+09,8.999999E+09]];
	LOCAL CONST Robtarget Tr_meulage_motif_2_P31 :=[[-48.94726953125,39.089984375,8.300712890625],[-1.55313807294348E-05,0.00588516465292523,0.0026390183776894,0.99997919987257],[0,0,0,0],[8.999999E+09,8.999999E+09,8.999999E+09,8.999999E+09,8.999999E+09,8.999999E+09]];
	LOCAL CONST Robtarget Tr_meulage_motif_2_P32 :=[[-48.176984375,40.15817578125,8.296322265625],[-1.55313807294348E-05,0.00588516465292523,0.0026390183776894,0.99997919987257],[0,0,0,0],[8.999999E+09,8.999999E+09,8.999999E+09,8.999999E+09,8.999999E+09,8.999999E+09]];
	LOCAL CONST Robtarget Tr_meulage_motif_2_P33 :=[[-47.82031640625,40.86633984375,8.29373828125],[-1.55313807294348E-05,0.00588516465292523,0.0026390183776894,0.99997919987257],[0,0,0,0],[8.999999E+09,8.999999E+09,8.999999E+09,8.999999E+09,8.999999E+09,8.999999E+09]];
	LOCAL CONST Robtarget Tr_meulage_motif_2_P34 :=[[-47.39837890625,42.04996484375,8.2897900390625],[-1.55313807294348E-05,0.00588516465292523,0.0026390183776894,0.99997919987257],[0,0,0,0],[8.999999E+09,8.999999E+09,8.999999E+09,8.999999E+09,8.999999E+09,8.999999E+09]];
	LOCAL CONST Robtarget Tr_meulage_motif_2_P35 :=[[-47.18200390625,42.90844921875,8.2871162109375],[-1.55313807294348E-05,0.00588516465292523,0.0026390183776894,0.99997919987257],[0,0,0,0],[8.999999E+09,8.999999E+09,8.999999E+09,8.999999E+09,8.999999E+09,8.999999E+09]];
	LOCAL CONST Robtarget Tr_meulage_motif_2_P36 :=[[-47.03002734375,43.8504296875,8.28436328125],[-1.55313807294348E-05,0.00588516465292523,0.0026390183776894,0.99997919987257],[0,0,0,0],[8.999999E+09,8.999999E+09,8.999999E+09,8.999999E+09,8.999999E+09,8.999999E+09]];
	LOCAL CONST Robtarget Tr_meulage_motif_2_P37 :=[[-46.976546875,44.83652734375,8.28170703125],[-1.55313807294348E-05,0.00588516465292523,0.0026390183776894,0.99997919987257],[0,0,0,0],[8.999999E+09,8.999999E+09,8.999999E+09,8.999999E+09,8.999999E+09,8.999999E+09]];
	LOCAL CONST Robtarget Tr_meulage_motif_2_P38 :=[[-46.9216875,45.83372265625,8.279017578125],[-1.55313807294348E-05,0.00588516465292523,0.0026390183776894,0.99997919987257],[0,0,0,0],[8.999999E+09,8.999999E+09,8.999999E+09,8.999999E+09,8.999999E+09,8.999999E+09]];
	LOCAL CONST Robtarget Tr_meulage_motif_2_P39 :=[[-46.9776640625,46.83215234375,8.2765615234375],[-1.55313807294348E-05,0.00588516465292523,0.0026390183776894,0.99997919987257],[0,0,0,0],[8.999999E+09,8.999999E+09,8.999999E+09,8.999999E+09,8.999999E+09,8.999999E+09]];
	LOCAL CONST Robtarget Tr_meulage_motif_2_P40 :=[[-47.033640625,47.830578125,8.27410546875],[-1.55313807294348E-05,0.00588516465292523,0.0026390183776894,0.99997919987257],[0,0,0,0],[8.999999E+09,8.999999E+09,8.999999E+09,8.999999E+09,8.999999E+09,8.999999E+09]];
	LOCAL CONST Robtarget Tr_meulage_motif_2_P41 :=[[-47.0896171875,48.8290078125,8.2716484375],[-1.55313807294348E-05,0.00588516465292523,0.0026390183776894,0.99997919987257],[0,0,0,0],[8.999999E+09,8.999999E+09,8.999999E+09,8.999999E+09,8.999999E+09,8.999999E+09]];
	LOCAL CONST Robtarget Tr_meulage_motif_2_P42 :=[[-47.14559375,49.8274375,8.2691923828125],[-1.55313807294348E-05,0.00588516465292523,0.0026390183776894,0.99997919987257],[0,0,0,0],[8.999999E+09,8.999999E+09,8.999999E+09,8.999999E+09,8.999999E+09,8.999999E+09]];
	LOCAL CONST Robtarget Tr_meulage_motif_2_P43 :=[[-47.2015703125,50.8258671875,8.2667353515625],[-1.55313807294348E-05,0.00588516465292523,0.0026390183776894,0.99997919987257],[0,0,0,0],[8.999999E+09,8.999999E+09,8.999999E+09,8.999999E+09,8.999999E+09,8.999999E+09]];
	LOCAL CONST Robtarget Tr_meulage_motif_2_P44 :=[[-47.257546875,51.824296875,8.264279296875],[-1.55313807294348E-05,0.00588516465292523,0.0026390183776894,0.99997919987257],[0,0,0,0],[8.999999E+09,8.999999E+09,8.999999E+09,8.999999E+09,8.999999E+09,8.999999E+09]];
	LOCAL CONST Robtarget Tr_meulage_motif_2_P45 :=[[-47.31352734375,52.8227265625,8.261822265625],[-1.55313807294348E-05,0.00588516465292523,0.0026390183776894,0.99997919987257],[0,0,0,0],[8.999999E+09,8.999999E+09,8.999999E+09,8.999999E+09,8.999999E+09,8.999999E+09]];
	LOCAL CONST Robtarget Tr_meulage_motif_2_P46 :=[[-47.36950390625,53.82115625,8.2593662109375],[-1.55313807294348E-05,0.00588516465292523,0.0026390183776894,0.99997919987257],[0,0,0,0],[8.999999E+09,8.999999E+09,8.999999E+09,8.999999E+09,8.999999E+09,8.999999E+09]];
	LOCAL CONST Robtarget Tr_meulage_motif_2_P47 :=[[-47.42548046875,54.81958203125,8.2569091796875],[-1.55313807294348E-05,0.00588516465292523,0.0026390183776894,0.99997919987257],[0,0,0,0],[8.999999E+09,8.999999E+09,8.999999E+09,8.999999E+09,8.999999E+09,8.999999E+09]];
	LOCAL CONST Robtarget Tr_meulage_motif_2_P48 :=[[-47.48145703125,55.81801171875,8.254453125],[-1.55313807294348E-05,0.00588516465292523,0.0026390183776894,0.99997919987257],[0,0,0,0],[8.999999E+09,8.999999E+09,8.999999E+09,8.999999E+09,8.999999E+09,8.999999E+09]];
	LOCAL CONST Robtarget Tr_meulage_motif_2_P49 :=[[-47.42659765625,56.81520703125,8.2517646484375],[-1.55313807294348E-05,0.00588516465292523,0.0026390183776894,0.99997919987257],[0,0,0,0],[8.999999E+09,8.999999E+09,8.999999E+09,8.999999E+09,8.999999E+09,8.999999E+09]];
	LOCAL CONST Robtarget Tr_meulage_motif_2_P50 :=[[-47.26872265625,57.7720390625,8.2489609375],[-1.55313807294348E-05,0.00588516465292523,0.0026390183776894,0.99997919987257],[0,0,0,0],[8.999999E+09,8.999999E+09,8.999999E+09,8.999999E+09,8.999999E+09,8.999999E+09]];
	LOCAL CONST Robtarget Tr_meulage_motif_2_P51 :=[[-47.0450390625,58.6386328125,8.2462509765625],[-1.55313807294348E-05,0.00588516465292523,0.0026390183776894,0.99997919987257],[0,0,0,0],[8.999999E+09,8.999999E+09,8.999999E+09,8.999999E+09,8.999999E+09,8.999999E+09]];
	LOCAL CONST Robtarget Tr_meulage_motif_2_P52 :=[[-46.7811875,59.3660390625,8.243814453125],[-1.55313807294348E-05,0.00588516465292523,0.0026390183776894,0.99997919987257],[0,0,0,0],[8.999999E+09,8.999999E+09,8.999999E+09,8.999999E+09,8.999999E+09,8.999999E+09]];
	LOCAL CONST Robtarget Tr_meulage_motif_2_P53 :=[[-46.1776015625,60.43596484375,8.2397734375],[-1.55313807294348E-05,0.00588516465292523,0.0026390183776894,0.99997919987257],[0,0,0,0],[8.999999E+09,8.999999E+09,8.999999E+09,8.999999E+09,8.999999E+09,8.999999E+09]];
	LOCAL CONST Robtarget Tr_meulage_motif_2_P54 :=[[-45.32756640625,61.38696875,8.2355166015625],[-1.55313807294348E-05,0.00588516465292523,0.0026390183776894,0.99997919987257],[0,0,0,0],[8.999999E+09,8.999999E+09,8.999999E+09,8.999999E+09,8.999999E+09,8.999999E+09]];
	LOCAL CONST Robtarget Tr_meulage_motif_2_P55 :=[[-44.313125,61.97964453125,8.231833984375],[-1.55313807294348E-05,0.00588516465292523,0.0026390183776894,0.99997919987257],[0,0,0,0],[8.999999E+09,8.999999E+09,8.999999E+09,8.999999E+09,8.999999E+09,8.999999E+09]];
	LOCAL CONST Robtarget Tr_meulage_motif_2_P56 :=[[-43.63133984375,62.2029375,8.229810546875],[-1.55313807294348E-05,0.00588516465292523,0.0026390183776894,0.99997919987257],[0,0,0,0],[8.999999E+09,8.999999E+09,8.999999E+09,8.999999E+09,8.999999E+09,8.999999E+09]];
	LOCAL CONST Robtarget Tr_meulage_motif_2_P57 :=[[-42.86612109375,62.30977734375,8.22791015625],[-1.55313807294348E-05,0.00588516465292523,0.0026390183776894,0.99997919987257],[0,0,0,0],[8.999999E+09,8.999999E+09,8.999999E+09,8.999999E+09,8.999999E+09,8.999999E+09]];
	LOCAL CONST Robtarget Tr_meulage_motif_2_P58 :=[[-42.09370703125,62.28603515625,8.22633203125],[-1.55313807294348E-05,0.00588516465292523,0.0026390183776894,0.99997919987257],[0,0,0,0],[8.999999E+09,8.999999E+09,8.999999E+09,8.999999E+09,8.999999E+09,8.999999E+09]];
	LOCAL CONST Robtarget Tr_meulage_motif_2_P59 :=[[-40.9637109375,61.9291328125,8.224853515625],[-1.55313807294348E-05,0.00588516465292523,0.0026390183776894,0.99997919987257],[0,0,0,0],[8.999999E+09,8.999999E+09,8.999999E+09,8.999999E+09,8.999999E+09,8.999999E+09]];
	LOCAL CONST Robtarget Tr_meulage_motif_2_P60 :=[[-40.35575,61.54825390625,8.2245458984375],[-1.55313807294348E-05,0.00588516465292523,0.0026390183776894,0.99997919987257],[0,0,0,0],[8.999999E+09,8.999999E+09,8.999999E+09,8.999999E+09,8.999999E+09,8.999999E+09]];
	LOCAL CONST Robtarget Tr_meulage_motif_2_P61 :=[[-39.420359375,60.71217578125,8.224716796875],[-1.55313807294348E-05,0.00588516465292523,0.0026390183776894,0.99997919987257],[0,0,0,0],[8.999999E+09,8.999999E+09,8.999999E+09,8.999999E+09,8.999999E+09,8.999999E+09]];
	LOCAL CONST Robtarget Tr_meulage_motif_2_P62 :=[[-38.9739140625,60.15059765625,8.2252177734375],[-1.55313807294348E-05,0.00588516465292523,0.0026390183776894,0.99997919987257],[0,0,0,0],[8.999999E+09,8.999999E+09,8.999999E+09,8.999999E+09,8.999999E+09,8.999999E+09]];
	LOCAL CONST Robtarget Tr_meulage_motif_2_P63 :=[[-38.36809765625,59.0648984375,8.2267314453125],[-1.55313807294348E-05,0.00588516465292523,0.0026390183776894,0.99997919987257],[0,0,0,0],[8.999999E+09,8.999999E+09,8.999999E+09,8.999999E+09,8.999999E+09,8.999999E+09]];
	LOCAL CONST Robtarget Tr_meulage_motif_2_P64 :=[[-38.02684765625,58.25714453125,8.2280908203125],[-1.55313807294348E-05,0.00588516465292523,0.0026390183776894,0.99997919987257],[0,0,0,0],[8.999999E+09,8.999999E+09,8.999999E+09,8.999999E+09,8.999999E+09,8.999999E+09]];
	LOCAL CONST Robtarget Tr_meulage_motif_2_P65 :=[[-37.77053125,57.33805078125,8.2299169921875],[-1.55313807294348E-05,0.00588516465292523,0.0026390183776894,0.99997919987257],[0,0,0,0],[8.999999E+09,8.999999E+09,8.999999E+09,8.999999E+09,8.999999E+09,8.999999E+09]];
	LOCAL CONST Robtarget Tr_meulage_motif_2_P66 :=[[-37.60716015625,56.364109375,8.2320830078125],[-1.55313807294348E-05,0.00588516465292523,0.0026390183776894,0.99997919987257],[0,0,0,0],[8.999999E+09,8.999999E+09,8.999999E+09,8.999999E+09,8.999999E+09,8.999999E+09]];
	LOCAL CONST Robtarget Tr_meulage_motif_2_P67 :=[[-37.4411796875,55.379296875,8.2342705078125],[-1.55313807294348E-05,0.00588516465292523,0.0026390183776894,0.99997919987257],[0,0,0,0],[8.999999E+09,8.999999E+09,8.999999E+09,8.999999E+09,8.999999E+09,8.999999E+09]];
	LOCAL CONST Robtarget Tr_meulage_motif_2_P68 :=[[-37.385203125,54.3808671875,8.2367265625],[-1.55313807294348E-05,0.00588516465292523,0.0026390183776894,0.99997919987257],[0,0,0,0],[8.999999E+09,8.999999E+09,8.999999E+09,8.999999E+09,8.999999E+09,8.999999E+09]];
	LOCAL CONST Robtarget Tr_meulage_motif_2_P69 :=[[-37.3292265625,53.3824375,8.23918359375],[-1.55313807294348E-05,0.00588516465292523,0.0026390183776894,0.99997919987257],[0,0,0,0],[8.999999E+09,8.999999E+09,8.999999E+09,8.999999E+09,8.999999E+09,8.999999E+09]];
	LOCAL CONST Robtarget Tr_meulage_motif_2_P70 :=[[-37.27325,52.3840078125,8.2416396484375],[-1.55313807294348E-05,0.00588516465292523,0.0026390183776894,0.99997919987257],[0,0,0,0],[8.999999E+09,8.999999E+09,8.999999E+09,8.999999E+09,8.999999E+09,8.999999E+09]];
	LOCAL CONST Robtarget Tr_meulage_motif_2_P71 :=[[-37.2172734375,51.385578125,8.2440966796875],[-1.55313807294348E-05,0.00588516465292523,0.0026390183776894,0.99997919987257],[0,0,0,0],[8.999999E+09,8.999999E+09,8.999999E+09,8.999999E+09,8.999999E+09,8.999999E+09]];
	LOCAL CONST Robtarget Tr_meulage_motif_2_P72 :=[[-37.161296875,50.38715234375,8.246552734375],[-1.55313807294348E-05,0.00588516465292523,0.0026390183776894,0.99997919987257],[0,0,0,0],[8.999999E+09,8.999999E+09,8.999999E+09,8.999999E+09,8.999999E+09,8.999999E+09]];
	LOCAL CONST Robtarget Tr_meulage_motif_2_P73 :=[[-37.1053203125,49.38872265625,8.249009765625],[-1.55313807294348E-05,0.00588516465292523,0.0026390183776894,0.99997919987257],[0,0,0,0],[8.999999E+09,8.999999E+09,8.999999E+09,8.999999E+09,8.999999E+09,8.999999E+09]];
	LOCAL CONST Robtarget Tr_meulage_motif_2_P74 :=[[-37.04934375,48.39029296875,8.2514658203125],[-1.55313807294348E-05,0.00588516465292523,0.0026390183776894,0.99997919987257],[0,0,0,0],[8.999999E+09,8.999999E+09,8.999999E+09,8.999999E+09,8.999999E+09,8.999999E+09]];
	LOCAL CONST Robtarget Tr_meulage_motif_2_P75 :=[[-36.9933671875,47.39186328125,8.2539228515625],[-1.55313807294348E-05,0.00588516465292523,0.0026390183776894,0.99997919987257],[0,0,0,0],[8.999999E+09,8.999999E+09,8.999999E+09,8.999999E+09,8.999999E+09,8.999999E+09]];
	LOCAL CONST Robtarget Tr_meulage_motif_2_P76 :=[[-36.937390625,46.39343359375,8.25637890625],[-1.55313807294348E-05,0.00588516465292523,0.0026390183776894,0.99997919987257],[0,0,0,0],[8.999999E+09,8.999999E+09,8.999999E+09,8.999999E+09,8.999999E+09,8.999999E+09]];
	LOCAL CONST Robtarget Tr_meulage_motif_2_P77 :=[[-36.8814140625,45.39500390625,8.2588359375],[-1.55313807294348E-05,0.00588516465292523,0.0026390183776894,0.99997919987257],[0,0,0,0],[8.999999E+09,8.999999E+09,8.999999E+09,8.999999E+09,8.999999E+09,8.999999E+09]];
	LOCAL CONST Robtarget Tr_meulage_motif_2_P78 :=[[-36.71543359375,44.41019140625,8.2610234375],[-1.55313807294348E-05,0.00588516465292523,0.0026390183776894,0.99997919987257],[0,0,0,0],[8.999999E+09,8.999999E+09,8.999999E+09,8.999999E+09,8.999999E+09,8.999999E+09]];
	LOCAL CONST Robtarget Tr_meulage_motif_2_P79 :=[[-36.45159375,43.477,8.2628701171875],[-1.55313807294348E-05,0.00588516465292523,0.0026390183776894,0.99997919987257],[0,0,0,0],[8.999999E+09,8.999999E+09,8.999999E+09,8.999999E+09,8.999999E+09,8.999999E+09]];
	LOCAL CONST Robtarget Tr_meulage_motif_2_P80 :=[[-36.1324453125,42.6408359375,8.264349609375],[-1.55313807294348E-05,0.00588516465292523,0.0026390183776894,0.99997919987257],[0,0,0,0],[8.999999E+09,8.999999E+09,8.999999E+09,8.999999E+09,8.999999E+09,8.999999E+09]];
	LOCAL CONST Robtarget Tr_meulage_motif_2_P81 :=[[-35.8149609375,41.90751953125,8.2655673828125],[-1.55313807294348E-05,0.00588516465292523,0.0026390183776894,0.99997919987257],[0,0,0,0],[8.999999E+09,8.999999E+09,8.999999E+09,8.999999E+09,8.999999E+09,8.999999E+09]];
	LOCAL CONST Robtarget Tr_meulage_motif_2_P82 :=[[-35.138171875,40.842671875,8.266876953125],[-1.55313807294348E-05,0.00588516465292523,0.0026390183776894,0.99997919987257],[0,0,0,0],[8.999999E+09,8.999999E+09,8.999999E+09,8.999999E+09,8.999999E+09,8.999999E+09]];
	LOCAL CONST Robtarget Tr_meulage_motif_2_P83 :=[[-34.19205078125,39.93749609375,8.267203125],[-1.55313807294348E-05,0.00588516465292523,0.0026390183776894,0.99997919987257],[0,0,0,0],[8.999999E+09,8.999999E+09,8.999999E+09,8.999999E+09,8.999999E+09,8.999999E+09]];
	LOCAL CONST Robtarget Tr_meulage_motif_2_P84 :=[[-33.07366015625,39.390109375,8.2662412109375],[-1.55313807294348E-05,0.00588516465292523,0.0026390183776894,0.99997919987257],[0,0,0,0],[8.999999E+09,8.999999E+09,8.999999E+09,8.999999E+09,8.999999E+09,8.999999E+09]];
	LOCAL CONST Robtarget Tr_meulage_motif_2_P85 :=[[-32.081353515625,39.27616015625,8.2644287109375],[-1.55313807294348E-05,0.00588516465292523,0.0026390183776894,0.99997919987257],[0,0,0,0],[8.999999E+09,8.999999E+09,8.999999E+09,8.999999E+09,8.999999E+09,8.999999E+09]];
	LOCAL CONST Robtarget Tr_meulage_motif_2_P86 :=[[-31.884376953125,39.41887890625,8.263642578125],[-1.55313807294348E-05,0.00588516465292523,0.0026390183776894,0.99997919987257],[0,0,0,0],[8.999999E+09,8.999999E+09,8.999999E+09,8.999999E+09,8.999999E+09,8.999999E+09]];
	LOCAL CONST Robtarget Tr_meulage_motif_2_P87 :=[[-31.166017578125,39.58271875,8.2616943359375],[-1.55313807294348E-05,0.00588516465292523,0.0026390183776894,0.99997919987257],[0,0,0,0],[8.999999E+09,8.999999E+09,8.999999E+09,8.999999E+09,8.999999E+09,8.999999E+09]];
	LOCAL CONST Robtarget Tr_meulage_motif_2_P88 :=[[-30.26887109375,40.31808203125,8.2578935546875],[-1.55313807294348E-05,0.00588516465292523,0.0026390183776894,0.99997919987257],[0,0,0,0],[8.999999E+09,8.999999E+09,8.999999E+09,8.999999E+09,8.999999E+09,8.999999E+09]];
	LOCAL CONST Robtarget Tr_meulage_motif_2_P89 :=[[-29.837,40.90079296875,8.2554736328125],[-1.55313807294348E-05,0.00588516465292523,0.0026390183776894,0.99997919987257],[0,0,0,0],[8.999999E+09,8.999999E+09,8.999999E+09,8.999999E+09,8.999999E+09,8.999999E+09]];
	LOCAL CONST Robtarget Tr_meulage_motif_2_P90 :=[[-29.37066796875,42.05901953125,8.25149609375],[-1.55313807294348E-05,0.00588516465292523,0.0026390183776894,0.99997919987257],[0,0,0,0],[8.999999E+09,8.999999E+09,8.999999E+09,8.999999E+09,8.999999E+09,8.999999E+09]];
	LOCAL CONST Robtarget Tr_meulage_motif_2_P91 :=[[-29.154291015625,42.91750390625,8.248822265625],[-1.55313807294348E-05,0.00588516465292523,0.0026390183776894,0.99997919987257],[0,0,0,0],[8.999999E+09,8.999999E+09,8.999999E+09,8.999999E+09,8.999999E+09,8.999999E+09]];
	LOCAL CONST Robtarget Tr_meulage_motif_2_P92 :=[[-29.0023125,43.859484375,8.2460703125],[-1.55313807294348E-05,0.00588516465292523,0.0026390183776894,0.99997919987257],[0,0,0,0],[8.999999E+09,8.999999E+09,8.999999E+09,8.999999E+09,8.999999E+09,8.999999E+09]];
	LOCAL CONST Robtarget Tr_meulage_motif_2_P93 :=[[-28.948833984375,44.84558203125,8.2434130859375],[-1.55313807294348E-05,0.00588516465292523,0.0026390183776894,0.99997919987257],[0,0,0,0],[8.999999E+09,8.999999E+09,8.999999E+09,8.999999E+09,8.999999E+09,8.999999E+09]];
	LOCAL CONST Robtarget Tr_meulage_motif_2_P94 :=[[-28.893974609375,45.8427734375,8.240724609375],[-1.55313807294348E-05,0.00588516465292523,0.0026390183776894,0.99997919987257],[0,0,0,0],[8.999999E+09,8.999999E+09,8.999999E+09,8.999999E+09,8.999999E+09,8.999999E+09]];
	LOCAL CONST Robtarget Tr_meulage_motif_2_P95 :=[[-28.949951171875,46.841203125,8.238267578125],[-1.55313807294348E-05,0.00588516465292523,0.0026390183776894,0.99997919987257],[0,0,0,0],[8.999999E+09,8.999999E+09,8.999999E+09,8.999999E+09,8.999999E+09,8.999999E+09]];
	LOCAL CONST Robtarget Tr_meulage_motif_2_P96 :=[[-29.005927734375,47.8396328125,8.2358115234375],[-1.55313807294348E-05,0.00588516465292523,0.0026390183776894,0.99997919987257],[0,0,0,0],[8.999999E+09,8.999999E+09,8.999999E+09,8.999999E+09,8.999999E+09,8.999999E+09]];
	LOCAL CONST Robtarget Tr_meulage_motif_2_P97 :=[[-29.061904296875,48.8380625,8.2333544921875],[-1.55313807294348E-05,0.00588516465292523,0.0026390183776894,0.99997919987257],[0,0,0,0],[8.999999E+09,8.999999E+09,8.999999E+09,8.999999E+09,8.999999E+09,8.999999E+09]];
	LOCAL CONST Robtarget Tr_meulage_motif_2_P98 :=[[-29.117880859375,49.8364921875,8.2308984375],[-1.55313807294348E-05,0.00588516465292523,0.0026390183776894,0.99997919987257],[0,0,0,0],[8.999999E+09,8.999999E+09,8.999999E+09,8.999999E+09,8.999999E+09,8.999999E+09]];
	LOCAL CONST Robtarget Tr_meulage_motif_2_P99 :=[[-29.173859375,50.834921875,8.22844140625],[-1.55313807294348E-05,0.00588516465292523,0.0026390183776894,0.99997919987257],[0,0,0,0],[8.999999E+09,8.999999E+09,8.999999E+09,8.999999E+09,8.999999E+09,8.999999E+09]];
	LOCAL CONST Robtarget Tr_meulage_motif_2_P100 :=[[-29.2298359375,51.8333515625,8.2259853515625],[-1.55313807294348E-05,0.00588516465292523,0.0026390183776894,0.99997919987257],[0,0,0,0],[8.999999E+09,8.999999E+09,8.999999E+09,8.999999E+09,8.999999E+09,8.999999E+09]];
	LOCAL CONST Robtarget Tr_meulage_motif_2_P101 :=[[-29.2858125,52.83177734375,8.223529296875],[-1.55313807294348E-05,0.00588516465292523,0.0026390183776894,0.99997919987257],[0,0,0,0],[8.999999E+09,8.999999E+09,8.999999E+09,8.999999E+09,8.999999E+09,8.999999E+09]];
	LOCAL CONST Robtarget Tr_meulage_motif_2_P102 :=[[-29.3417890625,53.83020703125,8.221072265625],[-1.55313807294348E-05,0.00588516465292523,0.0026390183776894,0.99997919987257],[0,0,0,0],[8.999999E+09,8.999999E+09,8.999999E+09,8.999999E+09,8.999999E+09,8.999999E+09]];
	LOCAL CONST Robtarget Tr_meulage_motif_2_P103 :=[[-29.397765625,54.82863671875,8.2186162109375],[-1.55313807294348E-05,0.00588516465292523,0.0026390183776894,0.99997919987257],[0,0,0,0],[8.999999E+09,8.999999E+09,8.999999E+09,8.999999E+09,8.999999E+09,8.999999E+09]];
	LOCAL CONST Robtarget Tr_meulage_motif_2_P104 :=[[-29.4537421875,55.82706640625,8.2161591796875],[-1.55313807294348E-05,0.00588516465292523,0.0026390183776894,0.99997919987257],[0,0,0,0],[8.999999E+09,8.999999E+09,8.999999E+09,8.999999E+09,8.999999E+09,8.999999E+09]];
	LOCAL CONST Robtarget Tr_meulage_motif_2_P105 :=[[-29.50971875,56.82549609375,8.213703125],[-1.55313807294348E-05,0.00588516465292523,0.0026390183776894,0.99997919987257],[0,0,0,0],[8.999999E+09,8.999999E+09,8.999999E+09,8.999999E+09,8.999999E+09,8.999999E+09]];
	LOCAL CONST Robtarget Tr_meulage_motif_2_P106 :=[[-29.5656953125,57.82392578125,8.21124609375],[-1.55313807294348E-05,0.00588516465292523,0.0026390183776894,0.99997919987257],[0,0,0,0],[8.999999E+09,8.999999E+09,8.999999E+09,8.999999E+09,8.999999E+09,8.999999E+09]];
	LOCAL CONST Robtarget Tr_meulage_motif_2_P107 :=[[-29.621671875,58.8223515625,8.2087900390625],[-1.55313807294348E-05,0.00588516465292523,0.0026390183776894,0.99997919987257],[0,0,0,0],[8.999999E+09,8.999999E+09,8.999999E+09,8.999999E+09,8.999999E+09,8.999999E+09]];
	LOCAL CONST Robtarget Tr_meulage_motif_2_P108 :=[[-29.677650390625,59.82078125,8.2063330078125],[-1.55313807294348E-05,0.00588516465292523,0.0026390183776894,0.99997919987257],[0,0,0,0],[8.999999E+09,8.999999E+09,8.999999E+09,8.999999E+09,8.999999E+09,8.999999E+09]];
	LOCAL CONST Robtarget Tr_meulage_motif_2_P109 :=[[-29.733626953125,60.8192109375,8.203876953125],[-1.55313807294348E-05,0.00588516465292523,0.0026390183776894,0.99997919987257],[0,0,0,0],[8.999999E+09,8.999999E+09,8.999999E+09,8.999999E+09,8.999999E+09,8.999999E+09]];
	LOCAL CONST Robtarget Tr_meulage_motif_2_P110 :=[[-29.789603515625,61.817640625,8.201419921875],[-1.55313807294348E-05,0.00588516465292523,0.0026390183776894,0.99997919987257],[0,0,0,0],[8.999999E+09,8.999999E+09,8.999999E+09,8.999999E+09,8.999999E+09,8.999999E+09]];
	LOCAL CONST Robtarget Tr_meulage_motif_2_P111 :=[[-29.845580078125,62.8160703125,8.1989638671875],[-1.55313807294348E-05,0.00588516465292523,0.0026390183776894,0.99997919987257],[0,0,0,0],[8.999999E+09,8.999999E+09,8.999999E+09,8.999999E+09,8.999999E+09,8.999999E+09]];
	LOCAL CONST Robtarget Tr_meulage_motif_2_P112 :=[[-29.901556640625,63.8145,8.1965078125],[-1.55313807294348E-05,0.00588516465292523,0.0026390183776894,0.99997919987257],[0,0,0,0],[8.999999E+09,8.999999E+09,8.999999E+09,8.999999E+09,8.999999E+09,8.999999E+09]];
	LOCAL CONST Robtarget Tr_meulage_motif_2_P113 :=[[-29.957533203125,64.81292578125,8.19405078125],[-1.55313807294348E-05,0.00588516465292523,0.0026390183776894,0.99997919987257],[0,0,0,0],[8.999999E+09,8.999999E+09,8.999999E+09,8.999999E+09,8.999999E+09,8.999999E+09]];
	LOCAL CONST Robtarget Tr_meulage_motif_2_P114 :=[[-30.013509765625,65.811359375,8.19159423828125],[-1.55313807294348E-05,0.00588516465292523,0.0026390183776894,0.99997919987257],[0,0,0,0],[8.999999E+09,8.999999E+09,8.999999E+09,8.999999E+09,8.999999E+09,8.999999E+09]];
	LOCAL CONST Robtarget Tr_meulage_motif_2_P115 :=[[-30.069486328125,66.8097890625,8.1891376953125],[-1.55313807294348E-05,0.00588516465292523,0.0026390183776894,0.99997919987257],[0,0,0,0],[8.999999E+09,8.999999E+09,8.999999E+09,8.999999E+09,8.999999E+09,8.999999E+09]];
	LOCAL CONST Robtarget Tr_meulage_motif_2_degg1 :=[[-30.187186353188,66.7570079646899,-1.8100303130677],[-1.55313807294348E-05,0.00588516465292523,0.0026390183776894,0.99997919987257],[0,0,0,0],[8.999999E+09,8.999999E+09,8.999999E+09,8.999999E+09,8.999999E+09,8.999999E+09]];
	LOCAL CONST Robtarget Tr_meulage_motif_2_degg2 :=[[-32.4234868293855,65.7541671062985,-191.794222472292],[-1.55313807294348E-05,0.00588516465292523,0.0026390183776894,0.99997919987257],[0,0,0,0],[8.999999E+09,8.999999E+09,8.999999E+09,8.999999E+09,8.999999E+09,8.999999E+09]];
	LOCAL CONST Robtarget Tr_meulage_bavure_App1 :=[[-198.321784326527,-218.718373899656,14.8136290565972],[0.632945220666498,-0.62138442776305,0.32352042528267,-0.329539489278516],[0,0,0,0],[8.999999E+09,8.999999E+09,8.999999E+09,8.999999E+09,8.999999E+09,8.999999E+09]];
	LOCAL CONST Robtarget Tr_meulage_bavure_App2 :=[[-42.6960470288263,-109.776345648108,18.3156814528299],[0.632945220666498,-0.62138442776305,0.32352042528267,-0.329539489278516],[0,0,0,0],[8.999999E+09,8.999999E+09,8.999999E+09,8.999999E+09,8.999999E+09,8.999999E+09]];
	LOCAL CONST Robtarget Tr_meulage_bavure_P0 :=[[-34.50521875,-104.0425546875,18.5],[0.632945220666498,-0.62138442776305,0.32352042528267,-0.329539489278516],[0,0,0,0],[8.999999E+09,8.999999E+09,8.999999E+09,8.999999E+09,8.999999E+09,8.999999E+09]];
	LOCAL CONST Robtarget Tr_meulage_bavure_P1 :=[[-36.25537109375,-101.5410625,18.5],[0.632883979764317,-0.621531474872828,0.32349548839717,-0.329404254506167],[0,0,0,0],[8.999999E+09,8.999999E+09,8.999999E+09,8.999999E+09,8.999999E+09,8.999999E+09]];
	LOCAL CONST Robtarget Tr_meulage_bavure_P2 :=[[-38.139921875,-98.94215625,18.5],[0.632708325756247,-0.621949080331058,0.323426231427532,-0.329021258915989],[0,0,0,0],[8.999999E+09,8.999999E+09,8.999999E+09,8.999999E+09,8.999999E+09,8.999999E+09]];
	LOCAL CONST Robtarget Tr_meulage_bavure_P3 :=[[-39.456421875,-96.8310703125,18.5],[0.632403334057888,-0.622606385125284,0.323350415979316,-0.328438458100901],[0,0,0,0],[8.999999E+09,8.999999E+09,8.999999E+09,8.999999E+09,8.999999E+09,8.999999E+09]];
	LOCAL CONST Robtarget Tr_meulage_bavure_P4 :=[[-40.31912109375,-95.707140625,18.5],[0.631935232607147,-0.623478272288081,0.323324535736219,-0.327710162133218],[0,0,0,0],[8.999999E+09,8.999999E+09,8.999999E+09,8.999999E+09,8.999999E+09,8.999999E+09]];
	LOCAL CONST Robtarget Tr_meulage_bavure_P5 :=[[-42.05346875,-93.2469140625,18.5],[0.63128804249874,-0.624503626277074,0.323408220468509,-0.326921628373355],[0,0,0,0],[8.999999E+09,8.999999E+09,8.999999E+09,8.999999E+09,8.999999E+09,8.999999E+09]];
	LOCAL CONST Robtarget Tr_meulage_bavure_P6 :=[[-42.05901953125,-93.2380703125,18.5],[0.630419658545921,-0.625626531269511,0.323690369241704,-0.326170265889909],[0,0,0,0],[8.999999E+09,8.999999E+09,8.999999E+09,8.999999E+09,8.999999E+09,8.999999E+09]];
	LOCAL CONST Robtarget Tr_meulage_bavure_P7 :=[[-42.0624375,-93.233109375,18.5],[0.629312156633084,-0.626761251269145,0.324252194087126,-0.32557189382844],[0,0,0,0],[8.999999E+09,8.999999E+09,8.999999E+09,8.999999E+09,8.999999E+09,8.999999E+09]];
	LOCAL CONST Robtarget Tr_meulage_bavure_P8 :=[[-43.30746484375,-91.437,18.5],[0.627931193144664,-0.627860789551483,0.325168826677205,-0.325205288667139],[0,0,0,0],[8.999999E+09,8.999999E+09,8.999999E+09,8.999999E+09,8.999999E+09,8.999999E+09]];
	LOCAL CONST Robtarget Tr_meulage_bavure_P9 :=[[-43.48547265625,-91.193203125,18.5],[0.626301978274772,-0.628893467277098,0.32643162831227,-0.325086497509043],[0,0,0,0],[8.999999E+09,8.999999E+09,8.999999E+09,8.999999E+09,8.999999E+09,8.999999E+09]];
	LOCAL CONST Robtarget Tr_meulage_bavure_P10 :=[[-43.8329765625,-90.7074140625,18.5],[0.624521686380947,-0.629870934742392,0.327913008505419,-0.32512817112574],[0,0,0,0],[8.999999E+09,8.999999E+09,8.999999E+09,8.999999E+09,8.999999E+09,8.999999E+09]];
	LOCAL CONST Robtarget Tr_meulage_bavure_P11 :=[[-46.2802734375,-87.065046875,18.5],[0.622693760568125,-0.630899353053157,0.329410662286844,-0.325126286907682],[0,0,0,0],[8.999999E+09,8.999999E+09,8.999999E+09,8.999999E+09,8.999999E+09,8.999999E+09]];
	LOCAL CONST Robtarget Tr_meulage_bavure_P12 :=[[-48.701234375,-83.8459296875,18.5],[0.620969389718729,-0.632053775566987,0.330686326706841,-0.324887049838866],[0,0,0,0],[8.999999E+09,8.999999E+09,8.999999E+09,8.999999E+09,8.999999E+09,8.999999E+09]];
	LOCAL CONST Robtarget Tr_meulage_bavure_P13 :=[[-48.953125,-83.46628125,18.5],[0.61942238860755,-0.633397541684085,0.331603865801889,-0.324287426314248],[0,0,0,0],[8.999999E+09,8.999999E+09,8.999999E+09,8.999999E+09,8.999999E+09,8.999999E+09]];
	LOCAL CONST Robtarget Tr_meulage_bavure_P14 :=[[-49.34295703125,-83.0005,18.5],[0.618074932679427,-0.634893794514995,0.33216059532165,-0.323361386370172],[0,0,0,0],[8.999999E+09,8.999999E+09,8.999999E+09,8.999999E+09,8.999999E+09,8.999999E+09]];
	LOCAL CONST Robtarget Tr_meulage_bavure_P15 :=[[-52.58416796875,-78.54625,18.5],[0.616870880517774,-0.636452667108397,0.332487710243091,-0.322258036109482],[0,0,0,0],[8.999999E+09,8.999999E+09,8.999999E+09,8.999999E+09,8.999999E+09,8.999999E+09]];
	LOCAL CONST Robtarget Tr_meulage_bavure_P16 :=[[-54.43963671875,-75.811328125,18.5],[0.615709373128981,-0.637981303017652,0.332775215248054,-0.321158031127398],[0,0,0,0],[8.999999E+09,8.999999E+09,8.999999E+09,8.999999E+09,8.999999E+09,8.999999E+09]];
	LOCAL CONST Robtarget Tr_meulage_bavure_P17 :=[[-55.94653125,-73.581234375,18.5],[0.614543081851257,-0.639390473618043,0.333148017458843,-0.320201532255073],[0,0,0,0],[8.999999E+09,8.999999E+09,8.999999E+09,8.999999E+09,8.999999E+09,8.999999E+09]];
	LOCAL CONST Robtarget Tr_meulage_bavure_P18 :=[[-56.7175,-72.5511328125,18.5],[0.613365006228656,-0.64065917757276,0.333632701349008,-0.319418859675629],[0,0,0,0],[8.999999E+09,8.999999E+09,8.999999E+09,8.999999E+09,8.999999E+09,8.999999E+09]];
	LOCAL CONST Robtarget Tr_meulage_bavure_P19 :=[[-58.32425,-70.2166015625,18.5],[0.612194669828632,-0.641825235638093,0.334179065283481,-0.318751322283968],[0,0,0,0],[8.999999E+09,8.999999E+09,8.999999E+09,8.999999E+09,8.999999E+09,8.999999E+09]];
	LOCAL CONST Robtarget Tr_meulage_bavure_P20 :=[[-59.67654296875,-68.4800703125,18.5],[0.611097076818949,-0.642923732424629,0.334682572012679,-0.318114779567842],[0,0,0,0],[8.999999E+09,8.999999E+09,8.999999E+09,8.999999E+09,8.999999E+09,8.999999E+09]];
	LOCAL CONST Robtarget Tr_meulage_bavure_P21 :=[[-60.60504296875,-67.1870234375,18.5],[0.610101630106608,-0.644018072017419,0.335059667536156,-0.317414150671936],[0,0,0,0],[8.999999E+09,8.999999E+09,8.999999E+09,8.999999E+09,8.999999E+09,8.999999E+09]];
	LOCAL CONST Robtarget Tr_meulage_bavure_P22 :=[[-61.737578125,-65.33940234375,18.5],[0.609244147509979,-0.645144732649506,0.335238468528823,-0.316583341125028],[0,0,0,0],[8.999999E+09,8.999999E+09,8.999999E+09,8.999999E+09,8.999999E+09,8.999999E+09]];
	LOCAL CONST Robtarget Tr_meulage_bavure_P23 :=[[-64.526125,-61.37187109375,18.5],[0.608531459745424,-0.646337648002134,0.335183410389439,-0.315577547799075],[0,0,0,0],[8.999999E+09,8.999999E+09,8.999999E+09,8.999999E+09,8.999999E+09,8.999999E+09]];
	LOCAL CONST Robtarget Tr_meulage_bavure_P24 :=[[-65.2424609375,-60.33608984375,18.5],[0.607958957037909,-0.647594263251933,0.334900350108076,-0.314403136527058],[0,0,0,0],[8.999999E+09,8.999999E+09,8.999999E+09,8.999999E+09,8.999999E+09,8.999999E+09]];
	LOCAL CONST Robtarget Tr_meulage_bavure_P25 :=[[-67.3720078125,-57.30157421875,18.5],[0.607496962969324,-0.64888291103812,0.334448644629912,-0.313117409051234],[0,0,0,0],[8.999999E+09,8.999999E+09,8.999999E+09,8.999999E+09,8.999999E+09,8.999999E+09]];
	LOCAL CONST Robtarget Tr_meulage_bavure_P26 :=[[-69.7112421875,-54.1526484375,18.5],[0.607062778487709,-0.650149217693107,0.333971867422404,-0.311839012117176],[0,0,0,0],[8.999999E+09,8.999999E+09,8.999999E+09,8.999999E+09,8.999999E+09,8.999999E+09]];
	LOCAL CONST Robtarget Tr_meulage_bavure_P27 :=[[-70.4522109375,-53.08770703125,18.5],[0.606569133365478,-0.651298187630351,0.333654313637705,-0.310740013883995],[0,0,0,0],[8.999999E+09,8.999999E+09,8.999999E+09,8.999999E+09,8.999999E+09,8.999999E+09]];
	LOCAL CONST Robtarget Tr_meulage_bavure_P28 :=[[-72.0042734375,-50.7165390625,18.5],[0.605940311755207,-0.652235138687233,0.333668671409874,-0.309985290249745],[0,0,0,0],[8.999999E+09,8.999999E+09,8.999999E+09,8.999999E+09,8.999999E+09,8.999999E+09]];
	LOCAL CONST Robtarget Tr_meulage_bavure_P29 :=[[-74.2776484375,-47.397734375,18.5],[0.605118741260492,-0.652916971919121,0.334124220373733,-0.309663918006165],[0,0,0,0],[8.999999E+09,8.999999E+09,8.999999E+09,8.999999E+09,8.999999E+09,8.999999E+09]];
	LOCAL CONST Robtarget Tr_meulage_bavure_P30 :=[[-76.1122421875,-44.90228125,18.5],[0.60412318957855,-0.653342412948291,0.335000629604431,-0.309763525000892],[0,0,0,0],[8.999999E+09,8.999999E+09,8.999999E+09,8.999999E+09,8.999999E+09,8.999999E+09]];
	LOCAL CONST Robtarget Tr_meulage_bavure_P31 :=[[-76.9116796875,-43.71819921875,18.5],[0.603013322709372,-0.65358592918878,0.336163598298416,-0.310152222272392],[0,0,0,0],[8.999999E+09,8.999999E+09,8.999999E+09,8.999999E+09,8.999999E+09,8.999999E+09]];
	LOCAL CONST Robtarget Tr_meulage_bavure_P32 :=[[-78.06771875,-42.11203125,18.5],[0.601903463632346,-0.653741483676987,0.337395626106271,-0.310642052001262],[0,0,0,0],[8.999999E+09,8.999999E+09,8.999999E+09,8.999999E+09,8.999999E+09,8.999999E+09]];
	LOCAL CONST Robtarget Tr_meulage_bavure_P33 :=[[-79.356046875,-40.19476171875,18.5],[0.600890753368103,-0.653916819335365,0.338490456628722,-0.311042290819611],[0,0,0,0],[8.999999E+09,8.999999E+09,8.999999E+09,8.999999E+09,8.999999E+09,8.999999E+09]];
	LOCAL CONST Robtarget Tr_meulage_bavure_P34 :=[[-80.90228125,-37.93805078125,18.5],[0.600047353406667,-0.654169958354234,0.339313944595638,-0.311240881407668],[0,0,0,0],[8.999999E+09,8.999999E+09,8.999999E+09,8.999999E+09,8.999999E+09,8.999999E+09]];
	LOCAL CONST Robtarget Tr_meulage_bavure_P35 :=[[-83.96096875,-33.4886171875,18.5],[0.599383948256652,-0.65450772975529,0.339848476744625,-0.311225845837394],[0,0,0,0],[8.999999E+09,8.999999E+09,8.999999E+09,8.999999E+09,8.999999E+09,8.999999E+09]];
	LOCAL CONST Robtarget Tr_meulage_bavure_P36 :=[[-86.207,-30.3984375,18.5],[0.598867271701993,-0.654886323559381,0.34017047124577,-0.311072249793386],[0,0,0,0],[8.999999E+09,8.999999E+09,8.999999E+09,8.999999E+09,8.999999E+09,8.999999E+09]];
	LOCAL CONST Robtarget Tr_meulage_bavure_P37 :=[[-86.3738984375,-30.156525390625,18.5],[0.598432633742364,-0.655237222165949,0.340414441490154,-0.310902836245306],[0,0,0,0],[8.999999E+09,8.999999E+09,8.999999E+09,8.999999E+09,8.999999E+09,8.999999E+09]];
	LOCAL CONST Robtarget Tr_meulage_bavure_P38 :=[[-86.5365,-29.930876953125,18.5],[0.598030367616643,-0.65547993671705,0.3407065281752,-0.310845288895484],[0,0,0,0],[8.999999E+09,8.999999E+09,8.999999E+09,8.999999E+09,8.999999E+09,8.999999E+09]];
	LOCAL CONST Robtarget Tr_meulage_bavure_P39 :=[[-91.5907265625,-22.702912109375,18.5],[0.597606186680911,-0.655569891725754,0.341149256167696,-0.310985767712305],[0,0,0,0],[8.999999E+09,8.999999E+09,8.999999E+09,8.999999E+09,8.999999E+09,8.999999E+09]];
	LOCAL CONST Robtarget Tr_meulage_bavure_P40 :=[[-95.7945859375,-16.7406015625,18.5],[0.597127810769619,-0.655480549144033,0.341803092586568,-0.311374811437241],[0,0,0,0],[8.999999E+09,8.999999E+09,8.999999E+09,8.999999E+09,8.999999E+09,8.999999E+09]];
	LOCAL CONST Robtarget Tr_meulage_bavure_P41 :=[[-97.1728203125,-14.758697265625,18.5],[0.59657647431841,-0.655206318061011,0.34269408080274,-0.31202877759193],[0,0,0,0],[8.999999E+09,8.999999E+09,8.999999E+09,8.999999E+09,8.999999E+09,8.999999E+09]];
	LOCAL CONST Robtarget Tr_meulage_bavure_P42 :=[[-99.23690625,-11.7934873046875,18.5],[0.595961646022882,-0.654753059765126,0.34380379542116,-0.312933055863242],[0,0,0,0],[8.999999E+09,8.999999E+09,8.999999E+09,8.999999E+09,8.999999E+09,8.999999E+09]];
	LOCAL CONST Robtarget Tr_meulage_bavure_P43 :=[[-100.3005078125,-10.2947080078125,18.5],[0.595304644480516,-0.654168592469388,0.345065407177034,-0.314015441748162],[0,0,0,0],[8.999999E+09,8.999999E+09,8.999999E+09,8.999999E+09,8.999999E+09,8.999999E+09]];
	LOCAL CONST Robtarget Tr_meulage_bavure_P44 :=[[-102.382171875,-7.283294921875,18.5],[0.594659081742485,-0.65353954118291,0.346343297224194,-0.315139596178407],[0,0,0,0],[8.999999E+09,8.999999E+09,8.999999E+09,8.999999E+09,8.999999E+09,8.999999E+09]];
	LOCAL CONST Robtarget Tr_meulage_bavure_P45 :=[[-105.067171875,-3.32406616210938,18.5],[0.594121751515497,-0.652983472306735,0.347428199351173,-0.316110068751375],[0,0,0,0],[8.999999E+09,8.999999E+09,8.999999E+09,8.999999E+09,8.999999E+09,8.999999E+09]];
	LOCAL CONST Robtarget Tr_meulage_bavure_P46 :=[[-106.182796875,-1.71005249023438,18.5],[0.593804004472896,-0.652634956563643,0.348083212217987,-0.316705691636782],[0,0,0,0],[8.999999E+09,8.999999E+09,8.999999E+09,8.999999E+09,8.999999E+09,8.999999E+09]];
	LOCAL CONST Robtarget Tr_meulage_bavure_P47 :=[[-107.4892578125,0.0113525390625,18.5],[0.593795836176519,-0.652605347691455,0.348116220358128,-0.316745737504888],[0,0,0,0],[8.999999E+09,8.999999E+09,8.999999E+09,8.999999E+09,8.999999E+09,8.999999E+09]];
	LOCAL CONST Robtarget Tr_meulage_bavure_P48 :=[[-108.8728046875,2.15350341796875,18.5],[0.594117001157093,-0.652944851730063,0.347464301353355,-0.316159087834485],[0,0,0,0],[8.999999E+09,8.999999E+09,8.999999E+09,8.999999E+09,8.999999E+09,8.999999E+09]];
	LOCAL CONST Robtarget Tr_meulage_bavure_P49 :=[[-109.9594140625,3.58087158203125,18.5],[0.594708626380983,-0.653609267814197,0.346228420436856,-0.315027706110485],[0,0,0,0],[8.999999E+09,8.999999E+09,8.999999E+09,8.999999E+09,8.999999E+09,8.999999E+09]];
	LOCAL CONST Robtarget Tr_meulage_bavure_P50 :=[[-111.015109375,5.03472900390625,18.5],[0.595452361253436,-0.654463919979732,0.344651104052349,-0.313574679140342],[0,0,0,0],[8.999999E+09,8.999999E+09,8.999999E+09,8.999999E+09,8.999999E+09,8.999999E+09]];
	LOCAL CONST Robtarget Tr_meulage_bavure_P51 :=[[-113.6263125,8.841216796875,18.5],[0.596189822063734,-0.655344323803907,0.343051091141757,-0.312085664829488],[0,0,0,0],[8.999999E+09,8.999999E+09,8.999999E+09,8.999999E+09,8.999999E+09,8.999999E+09]];
	LOCAL CONST Robtarget Tr_meulage_bavure_P52 :=[[-115.81525,11.865173828125,18.5],[0.596778316683267,-0.656108954947768,0.341716566023426,-0.310815811179534],[0,0,0,0],[8.999999E+09,8.999999E+09,8.999999E+09,8.999999E+09,8.999999E+09,8.999999E+09]];
	LOCAL CONST Robtarget Tr_meulage_bavure_P53 :=[[-117.2673984375,13.9100341796875,18.5],[0.597132454374457,-0.656671360205164,0.340826208934951,-0.309924268043125],[0,0,0,0],[8.999999E+09,8.999999E+09,8.999999E+09,8.999999E+09,8.999999E+09,8.999999E+09]];
	LOCAL CONST Robtarget Tr_meulage_bavure_P54 :=[[-119.4450078125,17.04684375,18.5],[0.597230448159599,-0.657011277629002,0.340427779653809,-0.309452580695925],[0,0,0,0],[8.999999E+09,8.999999E+09,8.999999E+09,8.999999E+09,8.999999E+09,8.999999E+09]];
	LOCAL CONST Robtarget Tr_meulage_bavure_P55 :=[[-120.2079453125,18.12109375,18.5],[0.59710816187658,-0.657168360166439,0.340447556918633,-0.309333235208665],[0,0,0,0],[8.999999E+09,8.999999E+09,8.999999E+09,8.999999E+09,8.999999E+09,8.999999E+09]];
	LOCAL CONST Robtarget Tr_meulage_bavure_P56 :=[[-121.735171875,20.31820703125,18.5],[0.596838374063617,-0.657220385488189,0.340733421072958,-0.309428595814566],[0,0,0,0],[8.999999E+09,8.999999E+09,8.999999E+09,8.999999E+09,8.999999E+09,8.999999E+09]];
	LOCAL CONST Robtarget Tr_meulage_bavure_P57 :=[[-122.5204453125,21.43795703125,18.5],[0.596524689485678,-0.657271678762582,0.341073180902616,-0.309550190437033],[0,0,0,0],[8.999999E+09,8.999999E+09,8.999999E+09,8.999999E+09,8.999999E+09,8.999999E+09]];
	LOCAL CONST Robtarget Tr_meulage_bavure_P58 :=[[-125.869265625,26.18765234375,18.5],[0.596286205821704,-0.65744736109882,0.341218939258172,-0.309475949990435],[0,0,0,0],[8.999999E+09,8.999999E+09,8.999999E+09,8.999999E+09,8.999999E+09,8.999999E+09]];
	LOCAL CONST Robtarget Tr_meulage_bavure_P59 :=[[-127.2953828125,28.190154296875,18.5],[0.59623476587238,-0.657880827754996,0.340924246088641,-0.308978282192135],[0,0,0,0],[8.999999E+09,8.999999E+09,8.999999E+09,8.999999E+09,8.999999E+09,8.999999E+09]];
	LOCAL CONST Robtarget Tr_meulage_bavure_P60 :=[[-128.377015625,29.816986328125,18.5],[0.596468477741069,-0.658661921116834,0.33999189144137,-0.307888522822877],[0,0,0,0],[8.999999E+09,8.999999E+09,8.999999E+09,8.999999E+09,8.999999E+09,8.999999E+09]];
	LOCAL CONST Robtarget Tr_meulage_bavure_P61 :=[[-129.95959375,32.144591796875,18.5],[0.597012272359429,-0.659798739430705,0.338375861955126,-0.306176005173509],[0,0,0,0],[8.999999E+09,8.999999E+09,8.999999E+09,8.999999E+09,8.999999E+09,8.999999E+09]];
	LOCAL CONST Robtarget Tr_meulage_bavure_P62 :=[[-130.98171875,33.4605703125,18.5],[0.597781060794813,-0.661209170549986,0.336236565807909,-0.303982249398433],[0,0,0,0],[8.999999E+09,8.999999E+09,8.999999E+09,8.999999E+09,8.999999E+09,8.999999E+09]];
	LOCAL CONST Robtarget Tr_meulage_bavure_P63 :=[[-132.65340625,35.93630859375,18.5],[0.598615454580956,-0.662697946992835,0.333926318222383,-0.301635844333463],[0,0,0,0],[8.999999E+09,8.999999E+09,8.999999E+09,8.999999E+09,8.999999E+09,8.999999E+09]];
	LOCAL CONST Robtarget Tr_meulage_bavure_P64 :=[[-134.014796875,37.658234375,18.5],[0.599310377221343,-0.664018241994726,0.331912468306553,-0.299567954620811],[0,0,0,0],[8.999999E+09,8.999999E+09,8.999999E+09,8.999999E+09,8.999999E+09,8.999999E+09]];
	LOCAL CONST Robtarget Tr_meulage_bavure_P65 :=[[-136.6314375,41.7326953125,18.5],[0.599670705772216,-0.664950880411586,0.330640990515676,-0.298180996492602],[0,0,0,0],[8.999999E+09,8.999999E+09,8.999999E+09,8.999999E+09,8.999999E+09,8.999999E+09]];
	LOCAL CONST Robtarget Tr_meulage_bavure_P66 :=[[-137.01296875,42.21615625,18.5],[0.599580064132328,-0.665354372828104,0.330396035446672,-0.297734386685037],[0,0,0,0],[8.999999E+09,8.999999E+09,8.999999E+09,8.999999E+09,8.999999E+09,8.999999E+09]];
	LOCAL CONST Robtarget Tr_meulage_bavure_P67 :=[[-138.251671875,43.93566796875,18.5],[0.599029029545236,-0.665198512792833,0.331221678001329,-0.298273968629982],[0,0,0,0],[8.999999E+09,8.999999E+09,8.999999E+09,8.999999E+09,8.999999E+09,8.999999E+09]];
	LOCAL CONST Robtarget Tr_meulage_bavure_P68 :=[[-138.676640625,44.54183984375,18.5],[0.598100163287863,-0.664569692416538,0.332931968657644,-0.299632479618223],[0,0,0,0],[8.999999E+09,8.999999E+09,8.999999E+09,8.999999E+09,8.999999E+09,8.999999E+09]];
	LOCAL CONST Robtarget Tr_meulage_bavure_P69 :=[[-139.993015625,46.53625390625,18.5],[0.596957691255225,-0.663622807626132,0.33517418485286,-0.301503814002182],[0,0,0,0],[8.999999E+09,8.999999E+09,8.999999E+09,8.999999E+09,8.999999E+09,8.999999E+09]];
	LOCAL CONST Robtarget Tr_meulage_bavure_P70 :=[[-140.4765625,47.19085546875,18.5],[0.595789329172218,-0.662552457637524,0.337537762992936,-0.303525245534405],[0,0,0,0],[8.999999E+09,8.999999E+09,8.999999E+09,8.999999E+09,8.999999E+09,8.999999E+09]];
	LOCAL CONST Robtarget Tr_meulage_bavure_P71 :=[[-142.1379375,49.5452265625,18.5],[0.594763910451553,-0.661541220696673,0.339657467621323,-0.305371755132334],[0,0,0,0],[8.999999E+09,8.999999E+09,8.999999E+09,8.999999E+09,8.999999E+09,8.999999E+09]];
	LOCAL CONST Robtarget Tr_meulage_bavure_P72 :=[[-144.997375,53.7170390625,18.5],[0.594011800491705,-0.660715215923588,0.341273026294225,-0.306819337473424],[0,0,0,0],[8.999999E+09,8.999999E+09,8.999999E+09,8.999999E+09,8.999999E+09,8.999999E+09]];
	LOCAL CONST Robtarget Tr_meulage_bavure_P73 :=[[-145.96559375,55.129578125,18.5],[0.593598229922964,-0.660141816859674,0.342256843208414,-0.307756683668355],[0,0,0,0],[8.999999E+09,8.999999E+09,8.999999E+09,8.999999E+09,8.999999E+09,8.999999E+09]];
	LOCAL CONST Robtarget Tr_meulage_bavure_P74 :=[[-148.7320625,59.15884375,18.5],[0.593531228716183,-0.659812615276968,0.342612708645521,-0.308195595579504],[0,0,0,0],[8.999999E+09,8.999999E+09,8.999999E+09,8.999999E+09,8.999999E+09,8.999999E+09]];
	LOCAL CONST Robtarget Tr_meulage_bavure_P75 :=[[-149.253296875,59.92758203125,18.5],[0.593768472754939,-0.659668464373728,0.342444191758035,-0.308234477961602],[0,0,0,0],[8.999999E+09,8.999999E+09,8.999999E+09,8.999999E+09,8.999999E+09,8.999999E+09]];
	LOCAL CONST Robtarget Tr_meulage_bavure_P76 :=[[-151.9951875,63.78527734375,18.5],[0.59422780218529,-0.659628482895347,0.341918664775805,-0.308018198068155],[0,0,0,0],[8.999999E+09,8.999999E+09,8.999999E+09,8.999999E+09,8.999999E+09,8.999999E+09]];
	LOCAL CONST Robtarget Tr_meulage_bavure_P77 :=[[-152.459640625,64.51675390625,18.5],[0.594826875141949,-0.65959621850579,0.34121594027224,-0.307710089606853],[0,0,0,0],[8.999999E+09,8.999999E+09,8.999999E+09,8.999999E+09,8.999999E+09,8.999999E+09]];
	LOCAL CONST Robtarget Tr_meulage_bavure_P78 :=[[-152.660875,64.828734375,18.5],[0.5954805186766,-0.659491806000569,0.340506002723438,-0.307455967260454],[0,0,0,0],[8.999999E+09,8.999999E+09,8.999999E+09,8.999999E+09,8.999999E+09,8.999999E+09]];
	LOCAL CONST Robtarget Tr_meulage_bavure_P79 :=[[-153.0655,65.33157421875,18.5],[0.596111329977794,-0.659259718781284,0.339929743365687,-0.307368955881796],[0,0,0,0],[8.999999E+09,8.999999E+09,8.999999E+09,8.999999E+09,8.999999E+09,8.999999E+09]];
	LOCAL CONST Robtarget Tr_meulage_bavure_P80 :=[[-153.870015625,66.477328125,18.5],[0.596676373514548,-0.658860459839608,0.339572652326005,-0.307523354465559],[0,0,0,0],[8.999999E+09,8.999999E+09,8.999999E+09,8.999999E+09,8.999999E+09,8.999999E+09]];
	LOCAL CONST Robtarget Tr_meulage_bavure_P81 :=[[-156.15909375,69.63159375,18.5],[0.597137416574098,-0.658300107814047,0.339475829118863,-0.307935115281265],[0,0,0,0],[8.999999E+09,8.999999E+09,8.999999E+09,8.999999E+09,8.999999E+09,8.999999E+09]];
	LOCAL CONST Robtarget Tr_meulage_bavure_P82 :=[[-156.8079375,70.52871875,18.5],[0.597486145436625,-0.657614688875268,0.339618257461223,-0.3085654974001],[0,0,0,0],[8.999999E+09,8.999999E+09,8.999999E+09,8.999999E+09,8.999999E+09,8.999999E+09]];
	LOCAL CONST Robtarget Tr_meulage_bavure_P83 :=[[-157.764546875,71.930875,18.5],[0.597735114897533,-0.65687217909503,0.339926995561405,-0.309323957103189],[0,0,0,0],[8.999999E+09,8.999999E+09,8.999999E+09,8.999999E+09,8.999999E+09,8.999999E+09]];
	LOCAL CONST Robtarget Tr_meulage_bavure_P84 :=[[-160.48378125,75.8304140625,18.5],[0.597906841314603,-0.656169809788429,0.340293955654821,-0.310078399080307],[0,0,0,0],[8.999999E+09,8.999999E+09,8.999999E+09,8.999999E+09,8.999999E+09,8.999999E+09]];
	LOCAL CONST Robtarget Tr_meulage_bavure_P85 :=[[-161.056296875,76.57678125,18.5],[0.598040294116642,-0.655602253648586,0.340594852752041,-0.31069058225603],[0,0,0,0],[8.999999E+09,8.999999E+09,8.999999E+09,8.999999E+09,8.999999E+09,8.999999E+09]];
	LOCAL CONST Robtarget Tr_meulage_bavure_P86 :=[[-161.71253125,77.5237109375,18.5],[0.598144939663674,-0.65526708754379,0.340740235449077,-0.311036600873157],[0,0,0,0],[8.999999E+09,8.999999E+09,8.999999E+09,8.999999E+09,8.999999E+09,8.999999E+09]];
	LOCAL CONST Robtarget Tr_meulage_bavure_P87 :=[[-165.005125,82.202515625,18.5],[0.598207060570518,-0.655237403836074,0.34068878584616,-0.311036024435133],[0,0,0,0],[8.999999E+09,8.999999E+09,8.999999E+09,8.999999E+09,8.999999E+09,8.999999E+09]];
	LOCAL CONST Robtarget Tr_meulage_bavure_P88 :=[[-166.360875,83.979671875,18.5],[0.598185789487163,-0.65554644446354,0.340463225672038,-0.31067251628012],[0,0,0,0],[8.999999E+09,8.999999E+09,8.999999E+09,8.999999E+09,8.999999E+09,8.999999E+09]];
	LOCAL CONST Robtarget Tr_meulage_bavure_P89 :=[[-167.265671875,85.3250703125,18.5],[0.597999003629962,-0.656202494717492,0.340154920175377,-0.309984044532287],[0,0,0,0],[8.999999E+09,8.999999E+09,8.999999E+09,8.999999E+09,8.999999E+09,8.999999E+09]];
	LOCAL CONST Robtarget Tr_meulage_bavure_P90 :=[[-170.548,90.1409921875,18.5],[0.597557344833269,-0.657182507650953,0.339888256273474,-0.309050715127464],[0,0,0,0],[8.999999E+09,8.999999E+09,8.999999E+09,8.999999E+09,8.999999E+09,8.999999E+09]];
	LOCAL CONST Robtarget Tr_meulage_bavure_P91 :=[[-170.825234375,90.531765625,18.5],[0.596762063398029,-0.65847041151179,0.339792707226161,-0.307949140229903],[0,0,0,0],[8.999999E+09,8.999999E+09,8.999999E+09,8.999999E+09,8.999999E+09,8.999999E+09]];
	LOCAL CONST Robtarget Tr_meulage_bavure_P92 :=[[-170.87184375,90.5961640625,18.5],[0.595534009584494,-0.660048261890834,0.339974903514295,-0.306745171736329],[0,0,0,0],[8.999999E+09,8.999999E+09,8.999999E+09,8.999999E+09,8.999999E+09,8.999999E+09]];
	LOCAL CONST Robtarget Tr_meulage_bavure_P93 :=[[-171.0745625,90.8849765625,18.5],[0.593833118997707,-0.661915907283534,0.340478053850282,-0.305457449267154],[0,0,0,0],[8.999999E+09,8.999999E+09,8.999999E+09,8.999999E+09,8.999999E+09,8.999999E+09]];
	LOCAL CONST Robtarget Tr_meulage_bavure_P94 :=[[-176.059796875,97.7628515625,18.5],[0.591620614594337,-0.664102410307015,0.341317272584138,-0.304065052985635],[0,0,0,0],[8.999999E+09,8.999999E+09,8.999999E+09,8.999999E+09,8.999999E+09,8.999999E+09]];
	LOCAL CONST Robtarget Tr_meulage_bavure_P95 :=[[-176.50803125,98.4534296875,18.5],[0.588838586633285,-0.666554677817608,0.342599325379323,-0.302654394682801],[0,0,0,0],[8.999999E+09,8.999999E+09,8.999999E+09,8.999999E+09,8.999999E+09,8.999999E+09]];
	LOCAL CONST Robtarget Tr_meulage_bavure_P96 :=[[-180.166390625,103.5433984375,18.5],[0.585361022822243,-0.669115088292593,0.344605423925628,-0.301470684114942],[0,0,0,0],[8.999999E+09,8.999999E+09,8.999999E+09,8.999999E+09,8.999999E+09,8.999999E+09]];
	LOCAL CONST Robtarget Tr_meulage_bavure_P97 :=[[-180.528640625,104.0284765625,18.5],[0.580889687174141,-0.67142024505449,0.348008456223147,-0.301084938618456],[0,0,0,0],[8.999999E+09,8.999999E+09,8.999999E+09,8.999999E+09,8.999999E+09,8.999999E+09]];
	LOCAL CONST Robtarget Tr_meulage_bavure_P98 :=[[-181.457046875,105.4288046875,18.5],[0.574926240522156,-0.672815939458741,0.353966460033863,-0.302466981239948],[0,0,0,0],[8.999999E+09,8.999999E+09,8.999999E+09,8.999999E+09,8.999999E+09,8.999999E+09]];
	LOCAL CONST Robtarget Tr_meulage_bavure_P99 :=[[-184.8405,110.2579921875,18.5],[0.566780272689404,-0.672366458608991,0.36403011833856,-0.306864042810726],[0,0,0,0],[8.999999E+09,8.999999E+09,8.999999E+09,8.999999E+09,8.999999E+09,8.999999E+09]];
	LOCAL CONST Robtarget Tr_meulage_bavure_P100 :=[[-186.633796875,112.5310390625,18.5],[0.555645207085081,-0.668898570437483,0.37983744313475,-0.315525946798239],[0,0,0,0],[8.999999E+09,8.999999E+09,8.999999E+09,8.999999E+09,8.999999E+09,8.999999E+09]];
	LOCAL CONST Robtarget Tr_meulage_bavure_P101 :=[[-187.07753125,113.0947578125,18.5],[0.54074230370267,-0.661177854152855,0.40255481222969,-0.329228232864185],[0,0,0,0],[8.999999E+09,8.999999E+09,8.999999E+09,8.999999E+09,8.999999E+09,8.999999E+09]];
	LOCAL CONST Robtarget Tr_meulage_bavure_P102 :=[[-189.769890625,116.24471875,18.5],[0.521468395262585,-0.648094686026429,0.43241981671612,-0.347932598067161],[0,0,0,0],[8.999999E+09,8.999999E+09,8.999999E+09,8.999999E+09,8.999999E+09,8.999999E+09]];
	LOCAL CONST Robtarget Tr_meulage_bavure_P103 :=[[-191.050109375,118.5003046875,18.5],[0.49759081140218,-0.6289098746854,0.468489103107169,-0.370666580906823],[0,0,0,0],[8.999999E+09,8.999999E+09,8.999999E+09,8.999999E+09,8.999999E+09,8.999999E+09]];
	LOCAL CONST Robtarget Tr_meulage_bavure_P104 :=[[-191.921640625,119.587796875,18.5],[0.469315482295981,-0.603416330498409,0.508894873492465,-0.395800098406018],[0,0,0,0],[8.999999E+09,8.999999E+09,8.999999E+09,8.999999E+09,8.999999E+09,8.999999E+09]];
	LOCAL CONST Robtarget Tr_meulage_bavure_P105 :=[[-192.65103125,121.89465625,18.5],[0.437208437185407,-0.571898210845011,0.551425818695895,-0.42155757063743],[0,0,0,0],[8.999999E+09,8.999999E+09,8.999999E+09,8.999999E+09,8.999999E+09,8.999999E+09]];
	LOCAL CONST Robtarget Tr_meulage_bavure_P106 :=[[-192.71134375,122.763671875,18.5],[0.402175503869621,-0.53514142526054,0.593871432866155,-0.446312939855921],[0,0,0,0],[8.999999E+09,8.999999E+09,8.999999E+09,8.999999E+09,8.999999E+09,8.999999E+09]];
	LOCAL CONST Robtarget Tr_meulage_bavure_P107 :=[[-192.4986875,124.0343359375,18.5],[0.365614821398725,-0.494710404884108,0.63404395724228,-0.468589028848874],[0,0,0,0],[8.999999E+09,8.999999E+09,8.999999E+09,8.999999E+09,8.999999E+09,8.999999E+09]];
	LOCAL CONST Robtarget Tr_meulage_bavure_P108 :=[[-192.22278125,124.8120703125,18.5],[0.329443062876933,-0.45306211842681,0.669975066510201,-0.487170807236566],[0,0,0,0],[8.999999E+09,8.999999E+09,8.999999E+09,8.999999E+09,8.999999E+09,8.999999E+09]];
	LOCAL CONST Robtarget Tr_meulage_bavure_P109 :=[[-191.719359375,125.9086640625,18.5],[0.295655941093229,-0.412974321864928,0.700422786849926,-0.501445603867322],[0,0,0,0],[8.999999E+09,8.999999E+09,8.999999E+09,8.999999E+09,8.999999E+09,8.999999E+09]];
	LOCAL CONST Robtarget Tr_meulage_bavure_P110 :=[[-190.484890625,127.3201015625,18.5],[0.265488382383767,-0.376349855463994,0.725315070754394,-0.511658825046564],[0,0,0,0],[8.999999E+09,8.999999E+09,8.999999E+09,8.999999E+09,8.999999E+09,8.999999E+09]];
	LOCAL CONST Robtarget Tr_meulage_bavure_P111 :=[[-188.100890625,129.1961328125,18.5],[0.239035075748094,-0.343577655091954,0.745516351875997,-0.518673304276518],[0,0,0,0],[8.999999E+09,8.999999E+09,8.999999E+09,8.999999E+09,8.999999E+09,8.999999E+09]];
	LOCAL CONST Robtarget Tr_meulage_bavure_P112 :=[[-187.80584375,129.442109375,18.5],[0.215625890724334,-0.313946133082754,0.762175351163864,-0.523480691955266],[0,0,0,0],[8.999999E+09,8.999999E+09,8.999999E+09,8.999999E+09,8.999999E+09,8.999999E+09]];
	LOCAL CONST Robtarget Tr_meulage_bavure_P113 :=[[-187.2263125,129.7951015625,18.5],[0.194597540926276,-0.286704487546466,0.776150773230508,-0.526803863975816],[0,0,0,0],[8.999999E+09,8.999999E+09,8.999999E+09,8.999999E+09,8.999999E+09,8.999999E+09]];
	LOCAL CONST Robtarget Tr_meulage_bavure_P114 :=[[-185.321328125,130.7360859375,18.5],[0.17601358321794,-0.262144282910263,0.787744633201968,-0.528921531346325],[0,0,0,0],[8.999999E+09,8.999999E+09,8.999999E+09,8.999999E+09,8.999999E+09,8.999999E+09]];
	LOCAL CONST Robtarget Tr_meulage_bavure_P115 :=[[-184.87846875,130.909671875,18.5],[0.160699690184432,-0.241689324955042,0.796882731730454,-0.529848838488124],[0,0,0,0],[8.999999E+09,8.999999E+09,8.999999E+09,8.999999E+09,8.999999E+09,8.999999E+09]];
	LOCAL CONST Robtarget Tr_meulage_bavure_P116 :=[[-182.19759375,131.7629375,18.5],[0.149776165236141,-0.227248538595029,0.803440673387063,-0.529535916044344],[0,0,0,0],[8.999999E+09,8.999999E+09,8.999999E+09,8.999999E+09,8.999999E+09,8.999999E+09]];
	LOCAL CONST Robtarget Tr_meulage_bavure_P117 :=[[-180.671046875,132.26075,18.5],[0.143958033339612,-0.220139503902019,0.807462998322851,-0.528032375710275],[0,0,0,0],[8.999999E+09,8.999999E+09,8.999999E+09,8.999999E+09,8.999999E+09,8.999999E+09]];
	LOCAL CONST Robtarget Tr_meulage_bavure_P118 :=[[-178.432359375,133.007328125,18.5],[0.143116371494313,-0.220374818361749,0.809193218550377,-0.525508305067018],[0,0,0,0],[8.999999E+09,8.999999E+09,8.999999E+09,8.999999E+09,8.999999E+09,8.999999E+09]];
	LOCAL CONST Robtarget Tr_meulage_bavure_P119 :=[[-176.241546875,134.23409375,18.5],[0.146269757438961,-0.226611987476445,0.809043311434971,-0.522207894820692],[0,0,0,0],[8.999999E+09,8.999999E+09,8.999999E+09,8.999999E+09,8.999999E+09,8.999999E+09]];
	LOCAL CONST Robtarget Tr_meulage_bavure_P120 :=[[-175.4986875,134.724640625,18.5],[0.151872574238044,-0.23655515160336,0.807566324413184,-0.518471805518875],[0,0,0,0],[8.999999E+09,8.999999E+09,8.999999E+09,8.999999E+09,8.999999E+09,8.999999E+09]];
	LOCAL CONST Robtarget Tr_meulage_bavure_P121 :=[[-174.037546875,135.877015625,18.5],[0.158275097231287,-0.247678808558221,0.805418465327965,-0.514689515238412],[0,0,0,0],[8.999999E+09,8.999999E+09,8.999999E+09,8.999999E+09,8.999999E+09,8.999999E+09]];
	LOCAL CONST Robtarget Tr_meulage_bavure_P122 :=[[-170.84828125,138.318484375,18.5],[0.164186295833996,-0.257969323867967,0.803216378828105,-0.511212418653618],[0,0,0,0],[8.999999E+09,8.999999E+09,8.999999E+09,8.999999E+09,8.999999E+09,8.999999E+09]];
	LOCAL CONST Robtarget Tr_meulage_bavure_P123 :=[[-169.0331875,139.750453125,18.5],[0.16887691388133,-0.266263563876064,0.80139466163973,-0.508282302274315],[0,0,0,0],[8.999999E+09,8.999999E+09,8.999999E+09,8.999999E+09,8.999999E+09,8.999999E+09]];
	LOCAL CONST Robtarget Tr_meulage_bavure_P124 :=[[-165.21640625,142.66290625,18.5],[0.172156276792755,-0.272243972672728,0.800143988076359,-0.50597928223346],[0,0,0,0],[8.999999E+09,8.999999E+09,8.999999E+09,8.999999E+09,8.999999E+09,8.999999E+09]];
	LOCAL CONST Robtarget Tr_meulage_bavure_P125 :=[[-162.545125,144.729890625,18.5],[0.174218719926156,-0.276200530464933,0.799429572163066,-0.504255355697248],[0,0,0,0],[8.999999E+09,8.999999E+09,8.999999E+09,8.999999E+09,8.999999E+09,8.999999E+09]];
	LOCAL CONST Robtarget Tr_meulage_bavure_P126 :=[[-161.79396875,145.33325,18.5],[0.17540643301786,-0.278672433676534,0.799110007019265,-0.502988523374459],[0,0,0,0],[8.999999E+09,8.999999E+09,8.999999E+09,8.999999E+09,8.999999E+09,8.999999E+09]];
	LOCAL CONST Robtarget Tr_meulage_bavure_P127 :=[[-157.648796875,148.643671875,18.5],[0.176067333314128,-0.280216125673027,0.799018340541412,-0.502044727619858],[0,0,0,0],[8.999999E+09,8.999999E+09,8.999999E+09,8.999999E+09,8.999999E+09,8.999999E+09]];
	LOCAL CONST Robtarget Tr_meulage_bavure_P128 :=[[-157.5999375,148.68215625,18.5],[0.176487679841728,-0.281285418939786,0.799004093780755,-0.501321324179959],[0,0,0,0],[8.999999E+09,8.999999E+09,8.999999E+09,8.999999E+09,8.999999E+09,8.999999E+09]];
	LOCAL CONST Robtarget Tr_meulage_bavure_P129 :=[[-157.53925,148.728578125,18.5],[0.17687001423023,-0.282206274801048,0.79895939107487,-0.500739960400991],[0,0,0,0],[8.999999E+09,8.999999E+09,8.999999E+09,8.999999E+09,8.999999E+09,8.999999E+09]];
	LOCAL CONST Robtarget Tr_meulage_bavure_P130 :=[[-153.9028125,151.59,18.5],[0.177334498509249,-0.283182699775763,0.79882450052005,-0.500239394245471],[0,0,0,0],[8.999999E+09,8.999999E+09,8.999999E+09,8.999999E+09,8.999999E+09,8.999999E+09]];
	LOCAL CONST Robtarget Tr_meulage_bavure_P131 :=[[-149.32909375,155.422265625,18.5],[0.177964883513843,-0.284355408640993,0.798555794736945,-0.499779095705857],[0,0,0,0],[8.999999E+09,8.999999E+09,8.999999E+09,8.999999E+09,8.999999E+09,8.999999E+09]];
	LOCAL CONST Robtarget Tr_meulage_bavure_P132 :=[[-147.76740625,156.74584375,18.5],[0.178814710914045,-0.285811560281624,0.798122921221062,-0.499336413444552],[0,0,0,0],[8.999999E+09,8.999999E+09,8.999999E+09,8.999999E+09,8.999999E+09,8.999999E+09]];
	LOCAL CONST Robtarget Tr_meulage_bavure_P133 :=[[-147.5309375,156.9646875,18.5],[0.179915058341048,-0.287600331606045,0.797506545662353,-0.498898717845547],[0,0,0,0],[8.999999E+09,8.999999E+09,8.999999E+09,8.999999E+09,8.999999E+09,8.999999E+09]];
	LOCAL CONST Robtarget Tr_meulage_bavure_P134 :=[[-144.975546875,159.054328125,18.5],[0.181266776955032,-0.289730753387558,0.79670846876057,-0.498451664576417],[0,0,0,0],[8.999999E+09,8.999999E+09,8.999999E+09,8.999999E+09,8.999999E+09,8.999999E+09]];
	LOCAL CONST Robtarget Tr_meulage_bavure_P135 :=[[-140.387140625,162.765984375,18.5],[0.182845445079206,-0.29216194074596,0.795740049540296,-0.498002728055729],[0,0,0,0],[8.999999E+09,8.999999E+09,8.999999E+09,8.999999E+09,8.999999E+09,8.999999E+09]];
	LOCAL CONST Robtarget Tr_meulage_bavure_P136 :=[[-136.16134375,166.2750625,18.5],[0.18460042239117,-0.294812492569045,0.7946292309555,-0.497566742848935],[0,0,0,0],[8.999999E+09,8.999999E+09,8.999999E+09,8.999999E+09,8.999999E+09,8.999999E+09]];
	LOCAL CONST Robtarget Tr_meulage_bavure_P137 :=[[-134.509671875,167.671328125,18.5],[0.186472435590399,-0.297590735655012,0.793411817591505,-0.497157392103786],[0,0,0,0],[8.999999E+09,8.999999E+09,8.999999E+09,8.999999E+09,8.999999E+09,8.999999E+09]];
	LOCAL CONST Robtarget Tr_meulage_bavure_P138 :=[[-129.37384375,172.14609375,18.5],[0.188424721528091,-0.300435232280521,0.792108465415598,-0.496788661845817],[0,0,0,0],[8.999999E+09,8.999999E+09,8.999999E+09,8.999999E+09,8.999999E+09,8.999999E+09]];
